KUKA KRL program: EPS_2_251727_MH2A_A_20260123013854.src

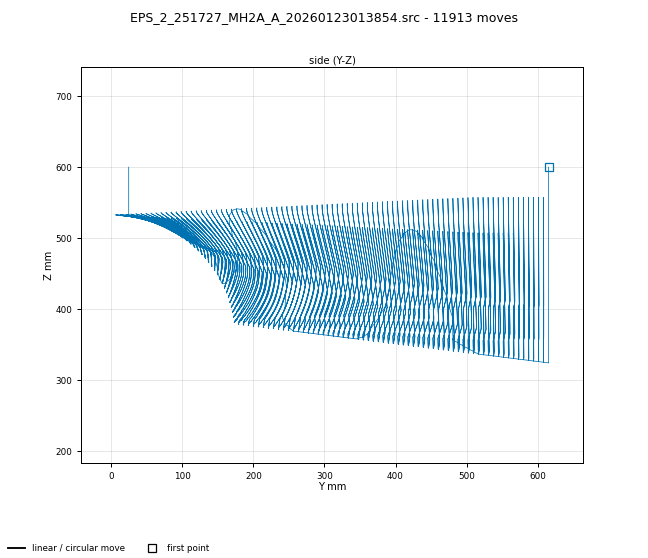
[picture p0: tool path of EPS_2_251727_MH2A_A_20260123013854.src, 11913 of 11915 moves have a stored position in this frame; points joined in program order, loops and branches not executed]
&ACCESS RVP
&REL 4
&COMMENT QRS 19112012
&PARAM EDITMASK = *
DEF PART()
EXT BAS (BAS_COMMAND :IN,REAL :IN )
INT I
BAS (#INITMOV,0 )

;KUKA QRS Post kuka4.cps  Date:22-06-2017 !

File_ID=2991

QRS_PRE_INIT()

;Init var - Until changes are made in qrs_pre_init
Outlet_Square_prg=0
Inlet_1_Square_prg=0
Inlet_2_Square_prg=0
Inlet_3_Square_prg=0
Inlet_4_Square_prg=0
Inlet_5_Square_prg=0

Outlet_1={X 0.000, Y 508.200, Z 408.000, B 0.000, E1 0.000 }
Inlet_1={X 0.000, Y 511.930, Z 358.000, B 0.000, E1 180.000 }
Outlet_1_type=299
Inlet_1_type=299
;QRS#1=Sidecore dimensions
;QRS#2=300-12" PVC SDR 35
;QRS#3=300-12" PVC SDR 35
;QRS#4=
;QRS#5=
;QRS#6=
;QRS#7=
;QRS#8=
;QRS#9=16M PSX
;QRS#10=16M PSX
;QRS#11=
;QRS#12=
;QRS#13=
;QRS#14=
;QRS#15=
;QRS#16=1220x127x838 2,75'
;QRS#17=EPS Height
;QRS#18=557,5
;QRS#19=*
;QRS#20= UPDATED VERSION 22-06-2017
;QRS#21=*
Outlet_Square=0150
Inlet_1_Square=0150
Inlet_2_Square=0
Inlet_3_Square=0
Inlet_4_Square=0
Inlet_5_Square=0
Mill_Square=1
Outlet_Square_Prg=206
Inlet_1_Square_prg=206

QRS_INIT()

$ADVANCE=5

; T1
PTP {E1 173.611,E2 173.611}
PTP {X 0,Y 615.501,A -85,B 0,C 180,E1 173.611,E2 173.611,E3 0,E4 0,E5 0,E6 0}
QRS_SPEED_INIT()
LIN {X 0,Y 615.501,Z 600,A -85,B 0,C 180,E1 173.611,E2 173.611,E3 0,E4 0,E5 0,E6 0} C_VEL
LIN {X 0,Y 615.501,Z 334.495,A -85,B 0,C 180,E1 173.611,E2 173.611} C_VEL
LIN {X 0,Y 615.501,Z 326.316,A -85,B 0,C 180,E1 173.611,E2 173.611} C_VEL
LIN {X 0,Y 615.486,Z 324.316,A -85,B 0,C 180,E1 173.425,E2 173.425} C_VEL
LIN {X 0,Y 615.496,Z 324.319,A -85,B 0,C 180,E1 170.801,E2 170.801} C_VEL
LIN {X 0,Y 615.493,Z 324.323,A -85,B 0,C 180,E1 168.139,E2 168.139} C_VEL
LIN {X 0,Y 615.481,Z 324.318,A -85,B 0,C 180,E1 165.451,E2 165.451} C_VEL
LIN {X 0,Y 615.494,Z 324.314,A -85,B 0,C 180,E1 162.73,E2 162.73} C_VEL
LIN {X 0,Y 615.494,Z 324.317,A -85,B 0,C 180,E1 159.967,E2 159.967} C_VEL
LIN {X 0,Y 615.493,Z 324.322,A -85,B 0,C 180,E1 157.156,E2 157.156} C_VEL
LIN {X 0,Y 615.5,Z 324.325,A -85,B 0,C 180,E1 154.285,E2 154.285} C_VEL
LIN {X 0,Y 615.479,Z 324.322,A -85,B 0,C 180,E1 151.552,E2 151.552} C_VEL
LIN {X 0,Y 615.487,Z 324.316,A -85,B 0,C 180,E1 148.915,E2 148.915} C_VEL
LIN {X 0,Y 615.49,Z 324.315,A -85,B 0,C 180,E1 145.978,E2 145.978} C_VEL
LIN {X 0,Y 615.487,Z 324.317,A -85,B 0,C 180,E1 143.064,E2 143.064} C_VEL
LIN {X 0,Y 615.495,Z 324.318,A -85,B 0,C 180,E1 140.25,E2 140.25} C_VEL
LIN {X 0,Y 615.487,Z 324.324,A -85,B 0,C 180,E1 137.647,E2 137.647} C_VEL
LIN {X 0,Y 615.487,Z 324.318,A -85,B 0,C 180,E1 134.931,E2 134.931} C_VEL
LIN {X 0,Y 615.481,Z 324.317,A -85,B 0,C 180,E1 132.079,E2 132.079} C_VEL
LIN {X 0,Y 615.496,Z 324.408,A -85,B 0,C 180,E1 131.473,E2 131.473} C_VEL
LIN {X 0,Y 615.484,Z 327.144,A -85,B 0,C 180,E1 128.905,E2 128.905} C_VEL
LIN {X 0,Y 615.494,Z 329.753,A -85,B 0,C 180,E1 126.425,E2 126.425} C_VEL
LIN {X 0,Y 615.496,Z 332.861,A -85,B 0,C 180,E1 123.535,E2 123.535} C_VEL
LIN {X 0,Y 615.48,Z 335.952,A -85,B 0,C 180,E1 120.92,E2 120.92} C_VEL
LIN {X 0,Y 615.491,Z 338.971,A -85,B 0,C 180,E1 118.451,E2 118.451} C_VEL
LIN {X 0,Y 615.499,Z 342.598,A -85,B 0,C 180,E1 115.571,E2 115.571} C_VEL
LIN {X 0,Y 615.482,Z 346.098,A -85,B 0,C 180,E1 112.845,E2 112.845} C_VEL
LIN {X 0,Y 615.484,Z 349.799,A -85,B 0,C 180,E1 110.033,E2 110.033} C_VEL
LIN {X 0,Y 615.478,Z 353.478,A -85,B 0,C 180,E1 107.271,E2 107.271} C_VEL
LIN {X 0,Y 615.481,Z 354.803,A -85,B 0,C 180,E1 106.298,E2 106.298} C_VEL
LIN {X 0,Y 615.497,Z 371.599,A -85,B 0,C 180,E1 106.003,E2 106.003} C_VEL
LIN {X 0,Y 615.49,Z 386.53,A -85,B 0,C 180,E1 105.608,E2 105.608} C_VEL
LIN {X 0,Y 615.48,Z 400.779,A -85,B 0,C 180,E1 105.099,E2 105.099} C_VEL
LIN {X 0,Y 615.482,Z 414.501,A -85,B 0,C 180,E1 104.473,E2 104.473} C_VEL
LIN {X 0,Y 615.496,Z 428.072,A -85,B 0,C 180,E1 103.706,E2 103.706} C_VEL
LIN {X 0,Y 615.496,Z 441.456,A -85,B 0,C 180,E1 102.782,E2 102.782} C_VEL
LIN {X 0,Y 615.495,Z 452.57,A -85,B 0,C 180,E1 101.861,E2 101.861} C_VEL
LIN {X 0,Y 615.493,Z 462.483,A -85,B 0,C 180,E1 100.89,E2 100.89} C_VEL
LIN {X 0,Y 615.495,Z 472.759,A -85,B 0,C 180,E1 99.696,E2 99.696} C_VEL
LIN {X 0,Y 615.49,Z 481.027,A -85,B 0,C 180,E1 98.537,E2 98.537} C_VEL
LIN {X 0,Y 615.491,Z 488.782,A -85,B 0,C 180,E1 97.216,E2 97.216} C_VEL
LIN {X 0,Y 615.499,Z 494.947,A -85,B 0,C 180,E1 95.899,E2 95.899} C_VEL
LIN {X 0,Y 615.489,Z 499.716,A -85,B 0,C 180,E1 94.585,E2 94.585} C_VEL
LIN {X 0,Y 615.491,Z 503.22,A -85,B 0,C 180,E1 93.273,E2 93.273} C_VEL
LIN {X 0,Y 615.5,Z 505.539,A -85,B 0,C 180,E1 91.963,E2 91.963} C_VEL
LIN {X 0,Y 615.491,Z 506.728,A -85,B 0,C 180,E1 90.655,E2 90.655} C_VEL
LIN {X 0,Y 615.492,Z 506.751,A -85,B 0,C 180,E1 89.346,E2 89.346} C_VEL
LIN {X 0,Y 615.5,Z 505.646,A -85,B 0,C 180,E1 88.037,E2 88.037} C_VEL
LIN {X 0,Y 615.494,Z 503.416,A -85,B 0,C 180,E1 86.727,E2 86.727} C_VEL
LIN {X 0,Y 615.49,Z 500.006,A -85,B 0,C 180,E1 85.416,E2 85.416} C_VEL
LIN {X 0,Y 615.499,Z 495.337,A -85,B 0,C 180,E1 84.102,E2 84.102} C_VEL
LIN {X 0,Y 615.49,Z 489.273,A -85,B 0,C 180,E1 82.785,E2 82.785} C_VEL
LIN {X 0,Y 615.493,Z 481.634,A -85,B 0,C 180,E1 81.464,E2 81.464} C_VEL
LIN {X 0,Y 615.496,Z 473.452,A -85,B 0,C 180,E1 80.304,E2 80.304} C_VEL
LIN {X 0,Y 615.495,Z 463.338,A -85,B 0,C 180,E1 79.109,E2 79.109} C_VEL
LIN {X 0,Y 615.497,Z 451.686,A -85,B 0,C 180,E1 77.973,E2 77.973} C_VEL
LIN {X 0,Y 615.498,Z 440.416,A -85,B 0,C 180,E1 77.051,E2 77.051} C_VEL
LIN {X 0,Y 615.498,Z 428.177,A -85,B 0,C 180,E1 76.211,E2 76.211} C_VEL
LIN {X 0,Y 615.49,Z 414.78,A -85,B 0,C 180,E1 75.451,E2 75.451} C_VEL
LIN {X 0,Y 615.478,Z 400.916,A -85,B 0,C 180,E1 74.816,E2 74.816} C_VEL
LIN {X 0,Y 615.496,Z 386.702,A -85,B 0,C 180,E1 74.308,E2 74.308} C_VEL
LIN {X 0,Y 615.494,Z 372.662,A -85,B 0,C 180,E1 73.932,E2 73.932} C_VEL
LIN {X 0,Y 615.483,Z 357.246,A -85,B 0,C 180,E1 73.652,E2 73.652} C_VEL
LIN {X 0,Y 615.483,Z 354.79,A -85,B 0,C 180,E1 73.603,E2 73.603} C_VEL
LIN {X 0,Y 615.487,Z 351.76,A -85,B 0,C 180,E1 71.354,E2 71.354} C_VEL
LIN {X 0,Y 615.485,Z 348.062,A -85,B 0,C 180,E1 68.568,E2 68.568} C_VEL
LIN {X 0,Y 615.48,Z 344.375,A -85,B 0,C 180,E1 65.728,E2 65.728} C_VEL
LIN {X 0,Y 615.48,Z 340.845,A -85,B 0,C 180,E1 62.957,E2 62.957} C_VEL
LIN {X 0,Y 615.477,Z 337.437,A -85,B 0,C 180,E1 60.207,E2 60.207} C_VEL
LIN {X 0,Y 615.493,Z 334.207,A -85,B 0,C 180,E1 57.543,E2 57.543} C_VEL
LIN {X 0,Y 615.497,Z 331.577,A -85,B 0,C 180,E1 55.186,E2 55.186} C_VEL
LIN {X 0,Y 615.493,Z 328.991,A -85,B 0,C 180,E1 52.759,E2 52.759} C_VEL
LIN {X 0,Y 615.49,Z 325.998,A -85,B 0,C 180,E1 49.911,E2 49.911} C_VEL
LIN {X 0,Y 615.497,Z 324.507,A -85,B 0,C 180,E1 48.527,E2 48.527} C_VEL
LIN {X 0,Y 615.491,Z 324.317,A -85,B 0,C 180,E1 45.851,E2 45.851} C_VEL
LIN {X 0,Y 615.483,Z 324.317,A -85,B 0,C 180,E1 43.047,E2 43.047} C_VEL
LIN {X 0,Y 615.481,Z 324.322,A -85,B 0,C 180,E1 40.607,E2 40.607} C_VEL
LIN {X 0,Y 615.485,Z 324.323,A -85,B 0,C 180,E1 38.012,E2 38.012} C_VEL
LIN {X 0,Y 615.481,Z 324.317,A -85,B 0,C 180,E1 35.616,E2 35.616} C_VEL
LIN {X 0,Y 615.489,Z 324.327,A -85,B 0,C 180,E1 33.236,E2 33.236} C_VEL
LIN {X 0,Y 615.49,Z 324.315,A -85,B 0,C 180,E1 30.92,E2 30.92} C_VEL
LIN {X 0,Y 615.479,Z 324.323,A -85,B 0,C 180,E1 28.45,E2 28.45} C_VEL
LIN {X 0,Y 615.498,Z 324.324,A -85,B 0,C 180,E1 25.715,E2 25.715} C_VEL
LIN {X 0,Y 615.494,Z 324.32,A -85,B 0,C 180,E1 22.844,E2 22.844} C_VEL
LIN {X 0,Y 615.493,Z 324.316,A -85,B 0,C 180,E1 20.033,E2 20.033} C_VEL
LIN {X 0,Y 615.493,Z 324.314,A -85,B 0,C 180,E1 17.27,E2 17.27} C_VEL
LIN {X 0,Y 615.481,Z 324.319,A -85,B 0,C 180,E1 14.549,E2 14.549} C_VEL
LIN {X 0,Y 615.492,Z 324.324,A -85,B 0,C 180,E1 11.861,E2 11.861} C_VEL
LIN {X 0,Y 615.496,Z 324.318,A -85,B 0,C 180,E1 9.199,E2 9.199} C_VEL
LIN {X 0,Y 615.487,Z 324.316,A -85,B 0,C 180,E1 6.557,E2 6.557} C_VEL
LIN {X 0,Y 615.48,Z 324.32,A -85,B 0,C 180,E1 3.929,E2 3.929} C_VEL
LIN {X 0,Y 615.495,Z 324.326,A -85,B 0,C 180,E1 1.309,E2 1.309} C_VEL
LIN {X 0,Y 615.487,Z 324.318,A -85,B 0,C 180,E1 -1.309,E2 -1.309} C_VEL
LIN {X 0,Y 615.478,Z 324.318,A -85,B 0,C 180,E1 -3.928,E2 -3.928} C_VEL
LIN {X 0,Y 615.486,Z 324.321,A -85,B 0,C 180,E1 -6.58,E2 -6.58} C_VEL
LIN {X 0,Y 615.489,Z 324.323,A -85,B 0,C 180,E1 -9.199,E2 -9.199} C_VEL
LIN {X 0,Y 615.477,Z 324.319,A -85,B 0,C 180,E1 -11.861,E2 -11.861} C_VEL
LIN {X 0,Y 615.481,Z 324.317,A -85,B 0,C 180,E1 -14.549,E2 -14.549} C_VEL
LIN {X 0,Y 615.493,Z 324.319,A -85,B 0,C 180,E1 -17.27,E2 -17.27} C_VEL
LIN {X 0,Y 615.493,Z 324.326,A -85,B 0,C 180,E1 -20.033,E2 -20.033} C_VEL
LIN {X 0,Y 615.483,Z 324.323,A -85,B 0,C 180,E1 -22.845,E2 -22.845} C_VEL
LIN {X 0,Y 615.476,Z 324.319,A -85,B 0,C 180,E1 -25.567,E2 -25.567} C_VEL
LIN {X 0,Y 615.491,Z 324.32,A -85,B 0,C 180,E1 -27.915,E2 -27.915} C_VEL
LIN {X 0,Y 615.492,Z 324.316,A -85,B 0,C 180,E1 -30.16,E2 -30.16} C_VEL
LIN {X 0,Y 615.477,Z 324.323,A -85,B 0,C 180,E1 -32.458,E2 -32.458} C_VEL
LIN {X 0,Y 615.491,Z 324.317,A -85,B 0,C 180,E1 -34.815,E2 -34.815} C_VEL
LIN {X 0,Y 615.479,Z 324.319,A -85,B 0,C 180,E1 -37.243,E2 -37.243} C_VEL
LIN {X 0,Y 615.483,Z 324.321,A -85,B 0,C 180,E1 -40.089,E2 -40.089} C_VEL
LIN {X 0,Y 615.477,Z 324.319,A -85,B 0,C 180,E1 -42.354,E2 -42.354} C_VEL
LIN {X 0,Y 615.479,Z 324.318,A -85,B 0,C 180,E1 -45.069,E2 -45.069} C_VEL
LIN {X 0,Y 615.485,Z 324.318,A -85,B 0,C 180,E1 -47.92,E2 -47.92} C_VEL
LIN {X 0,Y 615.499,Z 324.463,A -85,B 0,C 180,E1 -48.717,E2 -48.717} C_VEL
LIN {X 0,Y 615.482,Z 331.995,A -85,B 0,C 180,E1 -51.515,E2 -51.515} C_VEL
LIN {X 0,Y 615.48,Z 339.577,A -85,B 0,C 180,E1 -54.167,E2 -54.167} C_VEL
LIN {X 0,Y 615.485,Z 347.271,A -85,B 0,C 180,E1 -56.764,E2 -56.764} C_VEL
LIN {X 0,Y 615.496,Z 355.427,A -85,B 0,C 180,E1 -59.462,E2 -59.462} C_VEL
LIN {X 0,Y 615.495,Z 364.738,A -85,B 0,C 180,E1 -62.455,E2 -62.455} C_VEL
LIN {X 0,Y 615.493,Z 374.043,A -85,B 0,C 180,E1 -65.369,E2 -65.369} C_VEL
LIN {X 0,Y 615.489,Z 383.349,A -85,B 0,C 180,E1 -68.217,E2 -68.217} C_VEL
LIN {X 0,Y 615.484,Z 392.643,A -85,B 0,C 180,E1 -71.009,E2 -71.009} C_VEL
LIN {X 0,Y 615.488,Z 401.469,A -85,B 0,C 180,E1 -73.618,E2 -73.618} C_VEL
LIN {X 0,Y 615.493,Z 417.381,A -85,B 0,C 180,E1 -73.865,E2 -73.865} C_VEL
LIN {X 0,Y 615.497,Z 432.296,A -85,B 0,C 180,E1 -74.223,E2 -74.223} C_VEL
LIN {X 0,Y 615.478,Z 446.433,A -85,B 0,C 180,E1 -74.689,E2 -74.689} C_VEL
LIN {X 0,Y 615.496,Z 460.364,A -85,B 0,C 180,E1 -75.282,E2 -75.282} C_VEL
LIN {X 0,Y 615.499,Z 473.674,A -85,B 0,C 180,E1 -75.986,E2 -75.986} C_VEL
LIN {X 0,Y 615.498,Z 486.319,A -85,B 0,C 180,E1 -76.799,E2 -76.799} C_VEL
LIN {X 0,Y 615.496,Z 497.297,A -85,B 0,C 180,E1 -77.638,E2 -77.638} C_VEL
LIN {X 0,Y 615.497,Z 508.357,A -85,B 0,C 180,E1 -78.641,E2 -78.641} C_VEL
LIN {X 0,Y 615.496,Z 519.071,A -85,B 0,C 180,E1 -79.806,E2 -79.806} C_VEL
LIN {X 0,Y 615.495,Z 527.99,A -85,B 0,C 180,E1 -80.967,E2 -80.967} C_VEL
LIN {X 0,Y 615.492,Z 535.395,A -85,B 0,C 180,E1 -82.125,E2 -82.125} C_VEL
LIN {X 0,Y 615.491,Z 542.274,A -85,B 0,C 180,E1 -83.444,E2 -83.444} C_VEL
LIN {X 0,Y 615.491,Z 547.667,A -85,B 0,C 180,E1 -84.759,E2 -84.759} C_VEL
LIN {X 0,Y 615.491,Z 551.742,A -85,B 0,C 180,E1 -86.072,E2 -86.072} C_VEL
LIN {X 0,Y 615.496,Z 554.6,A -85,B 0,C 180,E1 -87.382,E2 -87.382} C_VEL
LIN {X 0,Y 615.493,Z 556.307,A -85,B 0,C 180,E1 -88.692,E2 -88.692} C_VEL
LIN {X 0,Y 615.491,Z 556.889,A -85,B 0,C 180,E1 -90,E2 -90} C_VEL
LIN {X 0,Y 615.493,Z 556.306,A -85,B 0,C 180,E1 -91.309,E2 -91.309} C_VEL
LIN {X 0,Y 615.496,Z 554.599,A -85,B 0,C 180,E1 -92.618,E2 -92.618} C_VEL
LIN {X 0,Y 615.491,Z 551.74,A -85,B 0,C 180,E1 -93.929,E2 -93.929} C_VEL
LIN {X 0,Y 615.491,Z 547.665,A -85,B 0,C 180,E1 -95.241,E2 -95.241} C_VEL
LIN {X 0,Y 615.491,Z 542.153,A -85,B 0,C 180,E1 -96.581,E2 -96.581} C_VEL
LIN {X 0,Y 615.492,Z 535.391,A -85,B 0,C 180,E1 -97.876,E2 -97.876} C_VEL
LIN {X 0,Y 615.495,Z 526.807,A -85,B 0,C 180,E1 -99.199,E2 -99.199} C_VEL
LIN {X 0,Y 615.494,Z 517.665,A -85,B 0,C 180,E1 -100.361,E2 -100.361} C_VEL
LIN {X 0,Y 615.497,Z 508.351,A -85,B 0,C 180,E1 -101.36,E2 -101.36} C_VEL
LIN {X 0,Y 615.496,Z 497.29,A -85,B 0,C 180,E1 -102.363,E2 -102.363} C_VEL
LIN {X 0,Y 615.498,Z 485.149,A -85,B 0,C 180,E1 -103.285,E2 -103.285} C_VEL
LIN {X 0,Y 615.498,Z 472.404,A -85,B 0,C 180,E1 -104.09,E2 -104.09} C_VEL
LIN {X 0,Y 615.496,Z 458.605,A -85,B 0,C 180,E1 -104.803,E2 -104.803} C_VEL
LIN {X 0,Y 615.48,Z 444.176,A -85,B 0,C 180,E1 -105.396,E2 -105.396} C_VEL
LIN {X 0,Y 615.496,Z 429.239,A -85,B 0,C 180,E1 -105.863,E2 -105.863} C_VEL
LIN {X 0,Y 615.491,Z 413.838,A -85,B 0,C 180,E1 -106.201,E2 -106.201} C_VEL
LIN {X 0,Y 615.488,Z 401.413,A -85,B 0,C 180,E1 -106.399,E2 -106.399} C_VEL
LIN {X 0,Y 615.484,Z 392.641,A -85,B 0,C 180,E1 -108.992,E2 -108.992} C_VEL
LIN {X 0,Y 615.489,Z 383.348,A -85,B 0,C 180,E1 -111.784,E2 -111.784} C_VEL
LIN {X 0,Y 615.493,Z 374.041,A -85,B 0,C 180,E1 -114.631,E2 -114.631} C_VEL
LIN {X 0,Y 615.494,Z 364.736,A -85,B 0,C 180,E1 -117.545,E2 -117.545} C_VEL
LIN {X 0,Y 615.496,Z 355.425,A -85,B 0,C 180,E1 -120.539,E2 -120.539} C_VEL
LIN {X 0,Y 615.485,Z 347.269,A -85,B 0,C 180,E1 -123.237,E2 -123.237} C_VEL
LIN {X 0,Y 615.48,Z 339.58,A -85,B 0,C 180,E1 -125.833,E2 -125.833} C_VEL
LIN {X 0,Y 615.485,Z 331.993,A -85,B 0,C 180,E1 -128.486,E2 -128.486} C_VEL
LIN {X 0,Y 615.498,Z 324.463,A -85,B 0,C 180,E1 -131.284,E2 -131.284} C_VEL
LIN {X 0,Y 615.491,Z 324.324,A -85,B 0,C 180,E1 -133.998,E2 -133.998} C_VEL
LIN {X 0,Y 615.483,Z 324.323,A -85,B 0,C 180,E1 -136.953,E2 -136.953} C_VEL
LIN {X 0,Y 615.482,Z 324.317,A -85,B 0,C 180,E1 -139.393,E2 -139.393} C_VEL
LIN {X 0,Y 615.493,Z 324.32,A -85,B 0,C 180,E1 -141.988,E2 -141.988} C_VEL
LIN {X 0,Y 615.487,Z 324.319,A -85,B 0,C 180,E1 -144.384,E2 -144.384} C_VEL
LIN {X 0,Y 615.481,Z 324.319,A -85,B 0,C 180,E1 -146.763,E2 -146.763} C_VEL
LIN {X 0,Y 615.493,Z 324.32,A -85,B 0,C 180,E1 -149.081,E2 -149.081} C_VEL
LIN {X 0,Y 615.478,Z 324.318,A -85,B 0,C 180,E1 -151.552,E2 -151.552} C_VEL
LIN {X 0,Y 615.477,Z 324.321,A -85,B 0,C 180,E1 -154.284,E2 -154.284} C_VEL
LIN {X 0,Y 615.474,Z 324.32,A -85,B 0,C 180,E1 -156.443,E2 -156.443} C_VEL
LIN {X 0,Y 615.498,Z 324.323,A -85,B 0,C 180,E1 -158.569,E2 -158.569} C_VEL
LIN {X 0,Y 615.486,Z 324.324,A -85,B 0,C 180,E1 -161.396,E2 -161.396} C_VEL
LIN {X 0,Y 615.482,Z 324.318,A -85,B 0,C 180,E1 -164.095,E2 -164.095} C_VEL
LIN {X 0,Y 615.494,Z 324.314,A -85,B 0,C 180,E1 -166.799,E2 -166.799} C_VEL
LIN {X 0,Y 615.494,Z 324.318,A -85,B 0,C 180,E1 -169.473,E2 -169.473} C_VEL
LIN {X 0,Y 615.49,Z 324.325,A -85,B 0,C 180,E1 -172.124,E2 -172.124} C_VEL
LIN {X 0,Y 615.487,Z 324.317,A -85,B 0,C 180,E1 -174.759,E2 -174.759} C_VEL
LIN {X 0,Y 615.491,Z 324.315,A -85,B 0,C 180,E1 -177.382,E2 -177.382} C_VEL
LIN {X 0,Y 615.486,Z 324.323,A -85,B 0,C 180,E1 -180,E2 -180} C_VEL
LIN {X 0,Y 615.496,Z 324.319,A -85,B 0,C 180,E1 -182.618,E2 -182.618} C_VEL
LIN {X 0,Y 615.487,Z 324.316,A -85,B 0,C 180,E1 -185.241,E2 -185.241} C_VEL
LIN {X 0,Y 615.486,Z 324.316,A -85,B 0,C 180,E1 -186.575,E2 -186.575} C_VEL
LIN {X 0,Y 614.812,Z 324.469,A -85,B 0,C 180,E1 -187.121,E2 -187.121} C_VEL
LIN {X 0,Y 611.984,Z 324.877,A -85,B 0,C 180,E1 -188.007,E2 -188.007} C_VEL
LIN {X 0,Y 609.595,Z 325.188,A -85,B 0,C 180,E1 -188.72,E2 -188.72} C_VEL
LIN {X 0,Y 608.556,Z 325.307,A -85,B 0,C 180,E1 -189.269,E2 -189.269} C_VEL
LIN {X 0,Y 608.464,Z 325.316,A -85,B 0,C 180,E1 -189.455,E2 -189.455} C_VEL
LIN {X 0,Y 608.466,Z 325.321,A -85,B 0,C 180,E1 -192,E2 -192} C_VEL
LIN {X 0,Y 608.474,Z 325.316,A -85,B 0,C 180,E1 -194.721,E2 -194.721} C_VEL
LIN {X 0,Y 608.458,Z 325.316,A -85,B 0,C 180,E1 -197.476,E2 -197.476} C_VEL
LIN {X 0,Y 608.461,Z 325.315,A -85,B 0,C 180,E1 -200.274,E2 -200.274} C_VEL
LIN {X 0,Y 608.462,Z 325.319,A -85,B 0,C 180,E1 -202.476,E2 -202.476} C_VEL
LIN {X 0,Y 608.458,Z 325.318,A -85,B 0,C 180,E1 -204.571,E2 -204.571} C_VEL
LIN {X 0,Y 608.485,Z 325.319,A -85,B 0,C 180,E1 -207.208,E2 -207.208} C_VEL
LIN {X 0,Y 608.47,Z 325.317,A -85,B 0,C 180,E1 -209.971,E2 -209.971} C_VEL
LIN {X 0,Y 608.459,Z 325.317,A -85,B 0,C 180,E1 -212.88,E2 -212.88} C_VEL
LIN {X 0,Y 608.443,Z 325.319,A -85,B 0,C 180,E1 -215.278,E2 -215.278} C_VEL
LIN {X 0,Y 608.467,Z 325.319,A -85,B 0,C 180,E1 -217.746,E2 -217.746} C_VEL
LIN {X 0,Y 608.448,Z 325.318,A -85,B 0,C 180,E1 -220.328,E2 -220.328} C_VEL
LIN {X 0,Y 608.45,Z 325.318,A -85,B 0,C 180,E1 -222.96,E2 -222.96} C_VEL
LIN {X 0,Y 608.46,Z 325.319,A -85,B 0,C 180,E1 -225.736,E2 -225.736} C_VEL
LIN {X 0,Y 608.461,Z 325.316,A -85,B 0,C 180,E1 -227.938,E2 -227.938} C_VEL
LIN {X 0,Y 608.445,Z 325.62,A -85,B 0,C 180,E1 -228.822,E2 -228.822} C_VEL
LIN {X 0,Y 608.438,Z 328.355,A -85,B 0,C 180,E1 -231.409,E2 -231.409} C_VEL
LIN {X 0,Y 608.451,Z 331.034,A -85,B 0,C 180,E1 -233.954,E2 -233.954} C_VEL
LIN {X 0,Y 608.456,Z 333.56,A -85,B 0,C 180,E1 -236.329,E2 -236.329} C_VEL
LIN {X 0,Y 608.449,Z 336.318,A -85,B 0,C 180,E1 -238.732,E2 -238.732} C_VEL
LIN {X 0,Y 608.427,Z 339.55,A -85,B 0,C 180,E1 -241.388,E2 -241.388} C_VEL
LIN {X 0,Y 608.428,Z 343.171,A -85,B 0,C 180,E1 -244.288,E2 -244.288} C_VEL
LIN {X 0,Y 608.413,Z 346.478,A -85,B 0,C 180,E1 -246.874,E2 -246.874} C_VEL
LIN {X 0,Y 608.427,Z 350.194,A -85,B 0,C 180,E1 -249.724,E2 -249.724} C_VEL
LIN {X 0,Y 608.41,Z 353.911,A -85,B 0,C 180,E1 -252.522,E2 -252.522} C_VEL
LIN {X 0,Y 608.441,Z 355.245,A -85,B 0,C 180,E1 -253.516,E2 -253.516} C_VEL
LIN {X 0,Y 608.671,Z 370.922,A -85,B 0,C 180,E1 -253.796,E2 -253.796} C_VEL
LIN {X 0,Y 608.641,Z 385.226,A -85,B 0,C 180,E1 -254.169,E2 -254.169} C_VEL
LIN {X 0,Y 608.614,Z 399.728,A -85,B 0,C 180,E1 -254.683,E2 -254.683} C_VEL
LIN {X 0,Y 608.572,Z 412.933,A -85,B 0,C 180,E1 -255.282,E2 -255.282} C_VEL
LIN {X 0,Y 608.565,Z 426.697,A -85,B 0,C 180,E1 -256.05,E2 -256.05} C_VEL
LIN {X 0,Y 608.548,Z 439.235,A -85,B 0,C 180,E1 -256.9,E2 -256.9} C_VEL
LIN {X 0,Y 608.522,Z 450.755,A -85,B 0,C 180,E1 -257.832,E2 -257.832} C_VEL
LIN {X 0,Y 608.483,Z 460.964,A -85,B 0,C 180,E1 -258.807,E2 -258.807} C_VEL
LIN {X 0,Y 608.48,Z 470.293,A -85,B 0,C 180,E1 -259.855,E2 -259.855} C_VEL
LIN {X 0,Y 608.447,Z 479.108,A -85,B 0,C 180,E1 -261.029,E2 -261.029} C_VEL
LIN {X 0,Y 608.457,Z 485.478,A -85,B 0,C 180,E1 -262.033,E2 -262.033} C_VEL
LIN {X 0,Y 608.445,Z 492.628,A -85,B 0,C 180,E1 -263.397,E2 -263.397} C_VEL
LIN {X 0,Y 608.435,Z 497.992,A -85,B 0,C 180,E1 -264.698,E2 -264.698} C_VEL
LIN {X 0,Y 608.432,Z 502.166,A -85,B 0,C 180,E1 -266.026,E2 -266.026} C_VEL
LIN {X 0,Y 608.421,Z 505.109,A -85,B 0,C 180,E1 -267.351,E2 -267.351} C_VEL
LIN {X 0,Y 608.444,Z 506.88,A -85,B 0,C 180,E1 -268.676,E2 -268.676} C_VEL
LIN {X 0,Y 608.432,Z 507.495,A -85,B 0,C 180,E1 -270,E2 -270} C_VEL
LIN {X 0,Y 608.446,Z 506.944,A -85,B 0,C 180,E1 -271.323,E2 -271.323} C_VEL
LIN {X 0,Y 608.424,Z 505.26,A -85,B 0,C 180,E1 -272.648,E2 -272.648} C_VEL
LIN {X 0,Y 608.431,Z 502.409,A -85,B 0,C 180,E1 -273.974,E2 -273.974} C_VEL
LIN {X 0,Y 608.435,Z 498.329,A -85,B 0,C 180,E1 -275.302,E2 -275.302} C_VEL
LIN {X 0,Y 608.445,Z 492.923,A -85,B 0,C 180,E1 -276.633,E2 -276.633} C_VEL
LIN {X 0,Y 608.456,Z 486.025,A -85,B 0,C 180,E1 -277.967,E2 -277.967} C_VEL
LIN {X 0,Y 608.466,Z 478.593,A -85,B 0,C 180,E1 -279.138,E2 -279.138} C_VEL
LIN {X 0,Y 608.476,Z 469.665,A -85,B 0,C 180,E1 -280.313,E2 -280.313} C_VEL
LIN {X 0,Y 608.495,Z 458.95,A -85,B 0,C 180,E1 -281.492,E2 -281.492} C_VEL
LIN {X 0,Y 608.513,Z 446.909,A -85,B 0,C 180,E1 -282.591,E2 -282.591} C_VEL
LIN {X 0,Y 608.543,Z 434.622,A -85,B 0,C 180,E1 -283.524,E2 -283.524} C_VEL
LIN {X 0,Y 608.579,Z 421.067,A -85,B 0,C 180,E1 -284.375,E2 -284.375} C_VEL
LIN {X 0,Y 608.592,Z 407.776,A -85,B 0,C 180,E1 -285.06,E2 -285.06} C_VEL
LIN {X 0,Y 608.615,Z 393.114,A -85,B 0,C 180,E1 -285.659,E2 -285.659} C_VEL
LIN {X 0,Y 608.664,Z 377.543,A -85,B 0,C 180,E1 -286.138,E2 -286.138} C_VEL
LIN {X 0,Y 608.67,Z 362.055,A -85,B 0,C 180,E1 -286.466,E2 -286.466} C_VEL
LIN {X 0,Y 608.428,Z 355.25,A -85,B 0,C 180,E1 -286.571,E2 -286.571} C_VEL
LIN {X 0,Y 608.42,Z 352.173,A -85,B 0,C 180,E1 -288.87,E2 -288.87} C_VEL
LIN {X 0,Y 608.41,Z 348.454,A -85,B 0,C 180,E1 -291.693,E2 -291.693} C_VEL
LIN {X 0,Y 608.417,Z 344.735,A -85,B 0,C 180,E1 -294.572,E2 -294.572} C_VEL
LIN {X 0,Y 608.427,Z 341.417,A -85,B 0,C 180,E1 -297.197,E2 -297.197} C_VEL
LIN {X 0,Y 608.442,Z 337.999,A -85,B 0,C 180,E1 -299.967,E2 -299.967} C_VEL
LIN {X 0,Y 608.435,Z 334.935,A -85,B 0,C 180,E1 -302.518,E2 -302.518} C_VEL
LIN {X 0,Y 608.448,Z 331.955,A -85,B 0,C 180,E1 -305.277,E2 -305.277} C_VEL
LIN {X 0,Y 608.454,Z 329.334,A -85,B 0,C 180,E1 -307.747,E2 -307.747} C_VEL
LIN {X 0,Y 608.442,Z 326.637,A -85,B 0,C 180,E1 -310.328,E2 -310.328} C_VEL
LIN {X 0,Y 608.47,Z 325.54,A -85,B 0,C 180,E1 -311.343,E2 -311.343} C_VEL
LIN {X 0,Y 608.468,Z 325.315,A -85,B 0,C 180,E1 -313.869,E2 -313.869} C_VEL
LIN {X 0,Y 608.467,Z 325.315,A -85,B 0,C 180,E1 -316.691,E2 -316.691} C_VEL
LIN {X 0,Y 608.452,Z 325.319,A -85,B 0,C 180,E1 -318.823,E2 -318.823} C_VEL
LIN {X 0,Y 608.472,Z 325.314,A -85,B 0,C 180,E1 -321.412,E2 -321.412} C_VEL
LIN {X 0,Y 608.479,Z 325.316,A -85,B 0,C 180,E1 -323.95,E2 -323.95} C_VEL
LIN {X 0,Y 608.448,Z 325.319,A -85,B 0,C 180,E1 -326.328,E2 -326.328} C_VEL
LIN {X 0,Y 608.477,Z 325.315,A -85,B 0,C 180,E1 -328.727,E2 -328.727} C_VEL
LIN {X 0,Y 608.472,Z 325.32,A -85,B 0,C 180,E1 -331.38,E2 -331.38} C_VEL
LIN {X 0,Y 608.448,Z 325.319,A -85,B 0,C 180,E1 -333.964,E2 -333.964} C_VEL
LIN {X 0,Y 608.467,Z 325.318,A -85,B 0,C 180,E1 -336.155,E2 -336.155} C_VEL
LIN {X 0,Y 608.468,Z 325.315,A -85,B 0,C 180,E1 -338.308,E2 -338.308} C_VEL
LIN {X 0,Y 608.453,Z 325.317,A -85,B 0,C 180,E1 -341.13,E2 -341.13} C_VEL
LIN {X 0,Y 608.458,Z 325.317,A -85,B 0,C 180,E1 -343.906,E2 -343.906} C_VEL
LIN {X 0,Y 608.468,Z 325.319,A -85,B 0,C 180,E1 -346.644,E2 -346.644} C_VEL
LIN {X 0,Y 608.467,Z 325.318,A -85,B 0,C 180,E1 -349.35,E2 -349.35} C_VEL
LIN {X 0,Y 608.472,Z 325.315,A -85,B 0,C 180,E1 -352.033,E2 -352.033} C_VEL
LIN {X 0,Y 608.467,Z 325.315,A -85,B 0,C 180,E1 -354.698,E2 -354.698} C_VEL
LIN {X 0,Y 608.486,Z 325.317,A -85,B 0,C 180,E1 -357.352,E2 -357.352} C_VEL
LIN {X 0,Y 608.474,Z 325.317,A -85,B 0,C 180,E1 -360,E2 -360} C_VEL
LIN {X 0,Y 608.481,Z 325.313,A -85,B 0,C 180,E1 -362.648,E2 -362.648} C_VEL
LIN {X 0,Y 608.47,Z 325.315,A -85,B 0,C 180,E1 -365.302,E2 -365.302} C_VEL
LIN {X 0,Y 608.482,Z 325.318,A -85,B 0,C 180,E1 -367.967,E2 -367.967} C_VEL
LIN {X 0,Y 608.473,Z 325.32,A -85,B 0,C 180,E1 -370.959,E2 -370.959} C_VEL
LIN {X 0,Y 608.471,Z 325.315,A -85,B 0,C 180,E1 -373.356,E2 -373.356} C_VEL
LIN {X 0,Y 608.46,Z 325.316,A -85,B 0,C 180,E1 -376.094,E2 -376.094} C_VEL
LIN {X 0,Y 608.457,Z 325.318,A -85,B 0,C 180,E1 -378.87,E2 -378.87} C_VEL
LIN {X 0,Y 608.478,Z 325.318,A -85,B 0,C 180,E1 -381.691,E2 -381.691} C_VEL
LIN {X 0,Y 608.46,Z 325.322,A -85,B 0,C 180,E1 -384.571,E2 -384.571} C_VEL
LIN {X 0,Y 608.455,Z 325.321,A -85,B 0,C 180,E1 -387.518,E2 -387.518} C_VEL
LIN {X 0,Y 608.47,Z 325.315,A -85,B 0,C 180,E1 -389.973,E2 -389.973} C_VEL
LIN {X 0,Y 608.454,Z 325.319,A -85,B 0,C 180,E1 -392.522,E2 -392.522} C_VEL
LIN {X 0,Y 608.446,Z 325.324,A -85,B 0,C 180,E1 -395.277,E2 -395.277} C_VEL
LIN {X 0,Y 608.473,Z 325.32,A -85,B 0,C 180,E1 -398.242,E2 -398.242} C_VEL
LIN {X 0,Y 608.464,Z 325.32,A -85,B 0,C 180,E1 -401.176,E2 -401.176} C_VEL
LIN {X 0,Y 608.474,Z 325.315,A -85,B 0,C 180,E1 -403.869,E2 -403.869} C_VEL
LIN {X 0,Y 608.482,Z 325.314,A -85,B 0,C 180,E1 -406.69,E2 -406.69} C_VEL
LIN {X 0,Y 608.48,Z 325.421,A -85,B 0,C 180,E1 -408.522,E2 -408.522} C_VEL
LIN {X 0,Y 608.506,Z 331.117,A -85,B 0,C 180,E1 -410.698,E2 -410.698} C_VEL
LIN {X 0,Y 608.516,Z 338.969,A -85,B 0,C 180,E1 -413.502,E2 -413.502} C_VEL
LIN {X 0,Y 608.504,Z 347.294,A -85,B 0,C 180,E1 -416.332,E2 -416.332} C_VEL
LIN {X 0,Y 608.507,Z 355.544,A -85,B 0,C 180,E1 -419.094,E2 -419.094} C_VEL
LIN {X 0,Y 608.476,Z 363.652,A -85,B 0,C 180,E1 -421.735,E2 -421.735} C_VEL
LIN {X 0,Y 608.475,Z 371.648,A -85,B 0,C 180,E1 -424.278,E2 -424.278} C_VEL
LIN {X 0,Y 608.464,Z 379.997,A -85,B 0,C 180,E1 -426.877,E2 -426.877} C_VEL
LIN {X 0,Y 608.468,Z 387.998,A -85,B 0,C 180,E1 -429.321,E2 -429.321} C_VEL
LIN {X 0,Y 608.449,Z 397.51,A -85,B 0,C 180,E1 -432.176,E2 -432.176} C_VEL
LIN {X 0,Y 608.462,Z 401.723,A -85,B 0,C 180,E1 -433.427,E2 -433.427} C_VEL
LIN {X 0,Y 608.678,Z 412.21,A -85,B 0,C 180,E1 -433.582,E2 -433.582} C_VEL
LIN {X 0,Y 608.656,Z 427.724,A -85,B 0,C 180,E1 -433.912,E2 -433.912} C_VEL
LIN {X 0,Y 608.629,Z 443.058,A -85,B 0,C 180,E1 -434.384,E2 -434.384} C_VEL
LIN {X 0,Y 608.615,Z 456.763,A -85,B 0,C 180,E1 -434.941,E2 -434.941} C_VEL
LIN {X 0,Y 608.591,Z 470.862,A -85,B 0,C 180,E1 -435.659,E2 -435.659} C_VEL
LIN {X 0,Y 608.543,Z 483.946,A -85,B 0,C 180,E1 -436.476,E2 -436.476} C_VEL
LIN {X 0,Y 608.512,Z 496.346,A -85,B 0,C 180,E1 -437.409,E2 -437.409} C_VEL
LIN {X 0,Y 608.496,Z 506.751,A -85,B 0,C 180,E1 -438.339,E2 -438.339} C_VEL
LIN {X 0,Y 608.477,Z 516.391,A -85,B 0,C 180,E1 -439.351,E2 -439.351} C_VEL
LIN {X 0,Y 608.476,Z 525.856,A -85,B 0,C 180,E1 -440.527,E2 -440.527} C_VEL
LIN {X 0,Y 608.456,Z 533.731,A -85,B 0,C 180,E1 -441.699,E2 -441.699} C_VEL
LIN {X 0,Y 608.441,Z 541.089,A -85,B 0,C 180,E1 -443.034,E2 -443.034} C_VEL
LIN {X 0,Y 608.45,Z 546.925,A -85,B 0,C 180,E1 -444.366,E2 -444.366} C_VEL
LIN {X 0,Y 608.427,Z 550.384,A -85,B 0,C 180,E1 -445.362,E2 -445.362} C_VEL
LIN {X 0,Y 608.421,Z 553.886,A -85,B 0,C 180,E1 -446.689,E2 -446.689} C_VEL
LIN {X 0,Y 608.444,Z 556.192,A -85,B 0,C 180,E1 -448.014,E2 -448.014} C_VEL
LIN {X 0,Y 608.436,Z 557.351,A -85,B 0,C 180,E1 -449.338,E2 -449.338} C_VEL
LIN {X 0,Y 608.436,Z 557.35,A -85,B 0,C 180,E1 -450.662,E2 -450.662} C_VEL
LIN {X 0,Y 608.444,Z 556.191,A -85,B 0,C 180,E1 -451.986,E2 -451.986} C_VEL
LIN {X 0,Y 608.421,Z 553.885,A -85,B 0,C 180,E1 -453.311,E2 -453.311} C_VEL
LIN {X 0,Y 608.427,Z 550.382,A -85,B 0,C 180,E1 -454.638,E2 -454.638} C_VEL
LIN {X 0,Y 608.437,Z 545.606,A -85,B 0,C 180,E1 -455.967,E2 -455.967} C_VEL
LIN {X 0,Y 608.457,Z 539.424,A -85,B 0,C 180,E1 -457.3,E2 -457.3} C_VEL
LIN {X 0,Y 608.468,Z 531.652,A -85,B 0,C 180,E1 -458.636,E2 -458.636} C_VEL
LIN {X 0,Y 608.471,Z 523.368,A -85,B 0,C 180,E1 -459.809,E2 -459.809} C_VEL
LIN {X 0,Y 608.493,Z 512.646,A -85,B 0,C 180,E1 -461.064,E2 -461.064} C_VEL
LIN {X 0,Y 608.522,Z 501.271,A -85,B 0,C 180,E1 -462.168,E2 -462.168} C_VEL
LIN {X 0,Y 608.547,Z 489.85,A -85,B 0,C 180,E1 -463.1,E2 -463.1} C_VEL
LIN {X 0,Y 608.563,Z 477.442,A -85,B 0,C 180,E1 -463.95,E2 -463.95} C_VEL
LIN {X 0,Y 608.602,Z 463.853,A -85,B 0,C 180,E1 -464.718,E2 -464.718} C_VEL
LIN {X 0,Y 608.6,Z 449.784,A -85,B 0,C 180,E1 -465.36,E2 -465.36} C_VEL
LIN {X 0,Y 608.661,Z 434.555,A -85,B 0,C 180,E1 -465.895,E2 -465.895} C_VEL
LIN {X 0,Y 608.69,Z 419.96,A -85,B 0,C 180,E1 -466.271,E2 -466.271} C_VEL
LIN {X 0,Y 608.673,Z 405.359,A -85,B 0,C 180,E1 -466.517,E2 -466.517} C_VEL
LIN {X 0,Y 608.458,Z 401.681,A -85,B 0,C 180,E1 -466.586,E2 -466.586} C_VEL
LIN {X 0,Y 608.462,Z 391.671,A -85,B 0,C 180,E1 -469.571,E2 -469.571} C_VEL
LIN {X 0,Y 608.479,Z 382.331,A -85,B 0,C 180,E1 -472.405,E2 -472.405} C_VEL
LIN {X 0,Y 608.461,Z 372.99,A -85,B 0,C 180,E1 -475.301,E2 -475.301} C_VEL
LIN {X 0,Y 608.472,Z 364.818,A -85,B 0,C 180,E1 -477.891,E2 -477.891} C_VEL
LIN {X 0,Y 608.496,Z 356.645,A -85,B 0,C 180,E1 -480.544,E2 -480.544} C_VEL
LIN {X 0,Y 608.516,Z 348.472,A -85,B 0,C 180,E1 -483.271,E2 -483.271} C_VEL
LIN {X 0,Y 608.49,Z 340.149,A -85,B 0,C 180,E1 -486.09,E2 -486.09} C_VEL
LIN {X 0,Y 608.507,Z 333.075,A -85,B 0,C 180,E1 -488.585,E2 -488.585} C_VEL
LIN {X 0,Y 608.565,Z 325.719,A -85,B 0,C 180,E1 -491.353,E2 -491.353} C_VEL
LIN {X 0,Y 608.465,Z 325.318,A -85,B 0,C 180,E1 -491.673,E2 -491.673} C_VEL
LIN {X 0,Y 608.466,Z 325.32,A -85,B 0,C 180,E1 -494.265,E2 -494.265} C_VEL
LIN {X 0,Y 608.449,Z 325.322,A -85,B 0,C 180,E1 -497.04,E2 -497.04} C_VEL
LIN {X 0,Y 608.454,Z 325.317,A -85,B 0,C 180,E1 -499.697,E2 -499.697} C_VEL
LIN {X 0,Y 608.472,Z 325.315,A -85,B 0,C 180,E1 -502.254,E2 -502.254} C_VEL
LIN {X 0,Y 608.482,Z 325.316,A -85,B 0,C 180,E1 -505.091,E2 -505.091} C_VEL
LIN {X 0,Y 608.465,Z 325.321,A -85,B 0,C 180,E1 -507.906,E2 -507.906} C_VEL
LIN {X 0,Y 608.472,Z 325.315,A -85,B 0,C 180,E1 -510.221,E2 -510.221} C_VEL
LIN {X 0,Y 608.488,Z 325.314,A -85,B 0,C 180,E1 -512.792,E2 -512.792} C_VEL
LIN {X 0,Y 608.484,Z 325.314,A -85,B 0,C 180,E1 -515.847,E2 -515.847} C_VEL
LIN {X 0,Y 608.478,Z 325.317,A -85,B 0,C 180,E1 -518.309,E2 -518.309} C_VEL
LIN {X 0,Y 608.472,Z 325.317,A -85,B 0,C 180,E1 -521.285,E2 -521.285} C_VEL
LIN {X 0,Y 608.46,Z 325.316,A -85,B 0,C 180,E1 -523.906,E2 -523.906} C_VEL
LIN {X 0,Y 608.472,Z 325.315,A -85,B 0,C 180,E1 -526.644,E2 -526.644} C_VEL
LIN {X 0,Y 608.472,Z 325.318,A -85,B 0,C 180,E1 -529.35,E2 -529.35} C_VEL
LIN {X 0,Y 608.481,Z 325.317,A -85,B 0,C 180,E1 -532.033,E2 -532.033} C_VEL
LIN {X 0,Y 608.466,Z 325.316,A -85,B 0,C 180,E1 -534.698,E2 -534.698} C_VEL
LIN {X 0,Y 608.482,Z 325.313,A -85,B 0,C 180,E1 -537.352,E2 -537.352} C_VEL
LIN {X 0,Y 608.477,Z 325.318,A -85,B 0,C 180,E1 -540,E2 -540} C_VEL
LIN {X 0,Y 608.487,Z 325.316,A -85,B 0,C 180,E1 -542.648,E2 -542.648} C_VEL
LIN {X 0,Y 608.468,Z 325.315,A -85,B 0,C 180,E1 -545.302,E2 -545.302} C_VEL
LIN {X 0,Y 608.473,Z 325.315,A -85,B 0,C 180,E1 -547.967,E2 -547.967} C_VEL
LIN {X 0,Y 608.464,Z 325.316,A -85,B 0,C 180,E1 -549.455,E2 -549.455} C_VEL
LIN {X 0,Y 607.778,Z 325.403,A -85,B 0,C 180,E1 -550.008,E2 -550.008} C_VEL
LIN {X 0,Y 604.925,Z 325.759,A -85,B 0,C 180,E1 -550.905,E2 -550.905} C_VEL
LIN {X 0,Y 602.526,Z 326.059,A -85,B 0,C 180,E1 -551.627,E2 -551.627} C_VEL
LIN {X 0,Y 601.497,Z 326.187,A -85,B 0,C 180,E1 -552.183,E2 -552.183} C_VEL
LIN {X 0,Y 601.412,Z 326.194,A -85,B 0,C 180,E1 -552.372,E2 -552.372} C_VEL
LIN {X 0,Y 601.43,Z 326.195,A -85,B 0,C 180,E1 -554.897,E2 -554.897} C_VEL
LIN {X 0,Y 601.438,Z 326.192,A -85,B 0,C 180,E1 -556.986,E2 -556.986} C_VEL
LIN {X 0,Y 601.412,Z 326.197,A -85,B 0,C 180,E1 -559.809,E2 -559.809} C_VEL
LIN {X 0,Y 601.415,Z 326.2,A -85,B 0,C 180,E1 -562.683,E2 -562.683} C_VEL
LIN {X 0,Y 601.408,Z 326.194,A -85,B 0,C 180,E1 -564.878,E2 -564.878} C_VEL
LIN {X 0,Y 601.421,Z 326.197,A -85,B 0,C 180,E1 -567.363,E2 -567.363} C_VEL
LIN {X 0,Y 601.432,Z 326.196,A -85,B 0,C 180,E1 -570.164,E2 -570.164} C_VEL
LIN {X 0,Y 601.418,Z 326.193,A -85,B 0,C 180,E1 -572.714,E2 -572.714} C_VEL
LIN {X 0,Y 601.401,Z 326.198,A -85,B 0,C 180,E1 -575.112,E2 -575.112} C_VEL
LIN {X 0,Y 601.437,Z 326.192,A -85,B 0,C 180,E1 -577.419,E2 -577.419} C_VEL
LIN {X 0,Y 601.415,Z 326.194,A -85,B 0,C 180,E1 -579.995,E2 -579.995} C_VEL
LIN {X 0,Y 601.412,Z 326.198,A -85,B 0,C 180,E1 -582.67,E2 -582.67} C_VEL
LIN {X 0,Y 601.429,Z 326.198,A -85,B 0,C 180,E1 -585.482,E2 -585.482} C_VEL
LIN {X 0,Y 601.428,Z 326.196,A -85,B 0,C 180,E1 -588.407,E2 -588.407} C_VEL
LIN {X 0,Y 601.384,Z 328.092,A -85,B 0,C 180,E1 -590.471,E2 -590.471} C_VEL
LIN {X 0,Y 601.37,Z 331.146,A -85,B 0,C 180,E1 -593.414,E2 -593.414} C_VEL
LIN {X 0,Y 601.384,Z 333.933,A -85,B 0,C 180,E1 -596.071,E2 -596.071} C_VEL
LIN {X 0,Y 601.37,Z 336.593,A -85,B 0,C 180,E1 -598.553,E2 -598.553} C_VEL
LIN {X 0,Y 601.342,Z 339.975,A -85,B 0,C 180,E1 -601.368,E2 -601.368} C_VEL
LIN {X 0,Y 601.346,Z 343.401,A -85,B 0,C 180,E1 -604.146,E2 -604.146} C_VEL
LIN {X 0,Y 601.334,Z 346.478,A -85,B 0,C 180,E1 -606.586,E2 -606.586} C_VEL
LIN {X 0,Y 601.345,Z 350.195,A -85,B 0,C 180,E1 -609.475,E2 -609.475} C_VEL
LIN {X 0,Y 601.31,Z 353.912,A -85,B 0,C 180,E1 -612.309,E2 -612.309} C_VEL
LIN {X 0,Y 601.344,Z 355.326,A -85,B 0,C 180,E1 -613.32,E2 -613.32} C_VEL
LIN {X 0,Y 601.881,Z 359.388,A -85,B 0,C 180,E1 -613.394,E2 -613.394} C_VEL
LIN {X 0,Y 601.838,Z 374.124,A -85,B 0,C 180,E1 -613.683,E2 -613.683} C_VEL
LIN {X 0,Y 601.767,Z 389.153,A -85,B 0,C 180,E1 -614.114,E2 -614.114} C_VEL
LIN {X 0,Y 601.742,Z 403.761,A -85,B 0,C 180,E1 -614.678,E2 -614.678} C_VEL
LIN {X 0,Y 601.652,Z 417.846,A -85,B 0,C 180,E1 -615.368,E2 -615.368} C_VEL
LIN {X 0,Y 601.621,Z 431.769,A -85,B 0,C 180,E1 -616.215,E2 -616.215} C_VEL
LIN {X 0,Y 601.531,Z 444.726,A -85,B 0,C 180,E1 -617.174,E2 -617.174} C_VEL
LIN {X 0,Y 601.489,Z 456.278,A -85,B 0,C 180,E1 -618.201,E2 -618.201} C_VEL
LIN {X 0,Y 601.43,Z 465.993,A -85,B 0,C 180,E1 -619.224,E2 -619.224} C_VEL
LIN {X 0,Y 601.429,Z 475.524,A -85,B 0,C 180,E1 -620.414,E2 -620.414} C_VEL
LIN {X 0,Y 601.378,Z 483.459,A -85,B 0,C 180,E1 -621.6,E2 -621.6} C_VEL
LIN {X 0,Y 601.368,Z 490.87,A -85,B 0,C 180,E1 -622.951,E2 -622.951} C_VEL
LIN {X 0,Y 601.373,Z 496.758,A -85,B 0,C 180,E1 -624.299,E2 -624.299} C_VEL
LIN {X 0,Y 601.327,Z 500.24,A -85,B 0,C 180,E1 -625.307,E2 -625.307} C_VEL
LIN {X 0,Y 601.336,Z 503.789,A -85,B 0,C 180,E1 -626.65,E2 -626.65} C_VEL
LIN {X 0,Y 601.343,Z 506.139,A -85,B 0,C 180,E1 -627.99,E2 -627.99} C_VEL
LIN {X 0,Y 601.334,Z 507.337,A -85,B 0,C 180,E1 -629.33,E2 -629.33} C_VEL
LIN {X 0,Y 601.335,Z 507.361,A -85,B 0,C 180,E1 -630.669,E2 -630.669} C_VEL
LIN {X 0,Y 601.343,Z 506.245,A -85,B 0,C 180,E1 -632.009,E2 -632.009} C_VEL
LIN {X 0,Y 601.339,Z 503.983,A -85,B 0,C 180,E1 -633.35,E2 -633.35} C_VEL
LIN {X 0,Y 601.328,Z 500.526,A -85,B 0,C 180,E1 -634.692,E2 -634.692} C_VEL
LIN {X 0,Y 601.358,Z 495.799,A -85,B 0,C 180,E1 -636.037,E2 -636.037} C_VEL
LIN {X 0,Y 601.365,Z 489.668,A -85,B 0,C 180,E1 -637.386,E2 -637.386} C_VEL
LIN {X 0,Y 601.389,Z 481.952,A -85,B 0,C 180,E1 -638.738,E2 -638.738} C_VEL
LIN {X 0,Y 601.428,Z 473.709,A -85,B 0,C 180,E1 -639.925,E2 -639.925} C_VEL
LIN {X 0,Y 601.443,Z 463.367,A -85,B 0,C 180,E1 -641.164,E2 -641.164} C_VEL
LIN {X 0,Y 601.503,Z 451.788,A -85,B 0,C 180,E1 -642.312,E2 -642.312} C_VEL
LIN {X 0,Y 601.557,Z 440.466,A -85,B 0,C 180,E1 -643.254,E2 -643.254} C_VEL
LIN {X 0,Y 601.623,Z 427.318,A -85,B 0,C 180,E1 -644.167,E2 -644.167} C_VEL
LIN {X 0,Y 601.673,Z 414.764,A -85,B 0,C 180,E1 -644.89,E2 -644.89} C_VEL
LIN {X 0,Y 601.731,Z 399.841,A -85,B 0,C 180,E1 -645.583,E2 -645.583} C_VEL
LIN {X 0,Y 601.816,Z 385.355,A -85,B 0,C 180,E1 -646.102,E2 -646.102} C_VEL
LIN {X 0,Y 601.866,Z 370.103,A -85,B 0,C 180,E1 -646.502,E2 -646.502} C_VEL
LIN {X 0,Y 601.76,Z 357.435,A -85,B 0,C 180,E1 -646.727,E2 -646.727} C_VEL
LIN {X 0,Y 601.338,Z 355.235,A -85,B 0,C 180,E1 -646.782,E2 -646.782} C_VEL
LIN {X 0,Y 601.313,Z 352.172,A -85,B 0,C 180,E1 -649.102,E2 -649.102} C_VEL
LIN {X 0,Y 601.315,Z 349.383,A -85,B 0,C 180,E1 -651.242,E2 -651.242} C_VEL
LIN {X 0,Y 601.342,Z 345.664,A -85,B 0,C 180,E1 -654.145,E2 -654.145} C_VEL
LIN {X 0,Y 601.34,Z 342.875,A -85,B 0,C 180,E1 -656.366,E2 -656.366} C_VEL
LIN {X 0,Y 601.341,Z 339.155,A -85,B 0,C 180,E1 -659.397,E2 -659.397} C_VEL
LIN {X 0,Y 601.339,Z 336.372,A -85,B 0,C 180,E1 -661.73,E2 -661.73} C_VEL
LIN {X 0,Y 601.381,Z 333.831,A -85,B 0,C 180,E1 -664.121,E2 -664.121} C_VEL
LIN {X 0,Y 601.367,Z 331.24,A -85,B 0,C 180,E1 -666.585,E2 -666.585} C_VEL
LIN {X 0,Y 601.384,Z 328.614,A -85,B 0,C 180,E1 -669.128,E2 -669.128} C_VEL
LIN {X 0,Y 601.396,Z 326.201,A -85,B 0,C 180,E1 -671.59,E2 -671.59} C_VEL
LIN {X 0,Y 601.449,Z 326.19,A -85,B 0,C 180,E1 -673.584,E2 -673.584} C_VEL
LIN {X 0,Y 601.428,Z 326.194,A -85,B 0,C 180,E1 -676.427,E2 -676.427} C_VEL
LIN {X 0,Y 601.413,Z 326.2,A -85,B 0,C 180,E1 -679.125,E2 -679.125} C_VEL
LIN {X 0,Y 601.421,Z 326.194,A -85,B 0,C 180,E1 -681.732,E2 -681.732} C_VEL
LIN {X 0,Y 601.408,Z 326.195,A -85,B 0,C 180,E1 -684.247,E2 -684.247} C_VEL
LIN {X 0,Y 601.417,Z 326.199,A -85,B 0,C 180,E1 -686.686,E2 -686.686} C_VEL
LIN {X 0,Y 601.433,Z 326.191,A -85,B 0,C 180,E1 -689.059,E2 -689.059} C_VEL
LIN {X 0,Y 601.431,Z 326.197,A -85,B 0,C 180,E1 -691.373,E2 -691.373} C_VEL
LIN {X 0,Y 601.405,Z 326.194,A -85,B 0,C 180,E1 -693.636,E2 -693.636} C_VEL
LIN {X 0,Y 601.421,Z 326.193,A -85,B 0,C 180,E1 -696.59,E2 -696.59} C_VEL
LIN {X 0,Y 601.427,Z 326.191,A -85,B 0,C 180,E1 -699.478,E2 -699.478} C_VEL
LIN {X 0,Y 601.402,Z 326.197,A -85,B 0,C 180,E1 -702.312,E2 -702.312} C_VEL
LIN {X 0,Y 601.416,Z 326.193,A -85,B 0,C 180,E1 -704.409,E2 -704.409} C_VEL
LIN {X 0,Y 601.421,Z 326.192,A -85,B 0,C 180,E1 -707.172,E2 -707.172} C_VEL
LIN {X 0,Y 601.43,Z 326.194,A -85,B 0,C 180,E1 -709.905,E2 -709.905} C_VEL
LIN {X 0,Y 601.439,Z 326.197,A -85,B 0,C 180,E1 -712.615,E2 -712.615} C_VEL
LIN {X 0,Y 601.421,Z 326.195,A -85,B 0,C 180,E1 -715.308,E2 -715.308} C_VEL
LIN {X 0,Y 601.419,Z 326.193,A -85,B 0,C 180,E1 -717.991,E2 -717.991} C_VEL
LIN {X 0,Y 601.45,Z 326.19,A -85,B 0,C 180,E1 -720.669,E2 -720.669} C_VEL
LIN {X 0,Y 601.435,Z 326.196,A -85,B 0,C 180,E1 -723.349,E2 -723.349} C_VEL
LIN {X 0,Y 601.407,Z 326.197,A -85,B 0,C 180,E1 -726.037,E2 -726.037} C_VEL
LIN {X 0,Y 601.414,Z 326.194,A -85,B 0,C 180,E1 -728.738,E2 -728.738} C_VEL
LIN {X 0,Y 601.435,Z 326.191,A -85,B 0,C 180,E1 -731.458,E2 -731.458} C_VEL
LIN {X 0,Y 601.418,Z 326.196,A -85,B 0,C 180,E1 -734.205,E2 -734.205} C_VEL
LIN {X 0,Y 601.433,Z 326.197,A -85,B 0,C 180,E1 -736.986,E2 -736.986} C_VEL
LIN {X 0,Y 601.408,Z 326.198,A -85,B 0,C 180,E1 -739.809,E2 -739.809} C_VEL
LIN {X 0,Y 601.41,Z 326.196,A -85,B 0,C 180,E1 -742.683,E2 -742.683} C_VEL
LIN {X 0,Y 601.405,Z 326.197,A -85,B 0,C 180,E1 -744.878,E2 -744.878} C_VEL
LIN {X 0,Y 601.422,Z 326.196,A -85,B 0,C 180,E1 -747.867,E2 -747.867} C_VEL
LIN {X 0,Y 601.447,Z 326.19,A -85,B 0,C 180,E1 -750.163,E2 -750.163} C_VEL
LIN {X 0,Y 601.416,Z 326.194,A -85,B 0,C 180,E1 -752.715,E2 -752.715} C_VEL
LIN {X 0,Y 601.414,Z 326.198,A -85,B 0,C 180,E1 -755.115,E2 -755.115} C_VEL
LIN {X 0,Y 601.434,Z 326.191,A -85,B 0,C 180,E1 -757.419,E2 -757.419} C_VEL
LIN {X 0,Y 601.409,Z 326.198,A -85,B 0,C 180,E1 -759.995,E2 -759.995} C_VEL
LIN {X 0,Y 601.408,Z 326.199,A -85,B 0,C 180,E1 -762.671,E2 -762.671} C_VEL
LIN {X 0,Y 601.424,Z 326.194,A -85,B 0,C 180,E1 -765.482,E2 -765.482} C_VEL
LIN {X 0,Y 601.44,Z 326.303,A -85,B 0,C 180,E1 -768.293,E2 -768.293} C_VEL
LIN {X 0,Y 601.557,Z 330.662,A -85,B 0,C 180,E1 -770.017,E2 -770.017} C_VEL
LIN {X 0,Y 601.536,Z 337.743,A -85,B 0,C 180,E1 -772.605,E2 -772.605} C_VEL
LIN {X 0,Y 601.528,Z 345.985,A -85,B 0,C 180,E1 -775.483,E2 -775.483} C_VEL
LIN {X 0,Y 601.526,Z 354.312,A -85,B 0,C 180,E1 -778.281,E2 -778.281} C_VEL
LIN {X 0,Y 601.496,Z 363.114,A -85,B 0,C 180,E1 -781.201,E2 -781.201} C_VEL
LIN {X 0,Y 601.435,Z 372.193,A -85,B 0,C 180,E1 -784.128,E2 -784.128} C_VEL
LIN {X 0,Y 601.431,Z 381.165,A -85,B 0,C 180,E1 -786.955,E2 -786.955} C_VEL
LIN {X 0,Y 601.423,Z 390.505,A -85,B 0,C 180,E1 -789.835,E2 -789.835} C_VEL
LIN {X 0,Y 601.389,Z 399.845,A -85,B 0,C 180,E1 -792.663,E2 -792.663} C_VEL
LIN {X 0,Y 601.388,Z 401.767,A -85,B 0,C 180,E1 -793.231,E2 -793.231} C_VEL
LIN {X 0,Y 601.864,Z 405.64,A -85,B 0,C 180,E1 -793.295,E2 -793.295} C_VEL
LIN {X 0,Y 601.855,Z 420.757,A -85,B 0,C 180,E1 -793.558,E2 -793.558} C_VEL
LIN {X 0,Y 601.807,Z 435.308,A -85,B 0,C 180,E1 -793.941,E2 -793.941} C_VEL
LIN {X 0,Y 601.737,Z 449.8,A -85,B 0,C 180,E1 -794.461,E2 -794.461} C_VEL
LIN {X 0,Y 601.691,Z 463.868,A -85,B 0,C 180,E1 -795.11,E2 -795.11} C_VEL
LIN {X 0,Y 601.613,Z 477.589,A -85,B 0,C 180,E1 -795.894,E2 -795.894} C_VEL
LIN {X 0,Y 601.57,Z 491.018,A -85,B 0,C 180,E1 -796.832,E2 -796.832} C_VEL
LIN {X 0,Y 601.513,Z 503.195,A -85,B 0,C 180,E1 -797.86,E2 -797.86} C_VEL
LIN {X 0,Y 601.437,Z 514.273,A -85,B 0,C 180,E1 -798.982,E2 -798.982} C_VEL
LIN {X 0,Y 601.427,Z 523.372,A -85,B 0,C 180,E1 -800.075,E2 -800.075} C_VEL
LIN {X 0,Y 601.388,Z 531.656,A -85,B 0,C 180,E1 -801.262,E2 -801.262} C_VEL
LIN {X 0,Y 601.365,Z 539.427,A -85,B 0,C 180,E1 -802.614,E2 -802.614} C_VEL
LIN {X 0,Y 601.357,Z 545.609,A -85,B 0,C 180,E1 -803.963,E2 -803.963} C_VEL
LIN {X 0,Y 601.33,Z 550.384,A -85,B 0,C 180,E1 -805.308,E2 -805.308} C_VEL
LIN {X 0,Y 601.337,Z 553.887,A -85,B 0,C 180,E1 -806.65,E2 -806.65} C_VEL
LIN {X 0,Y 601.343,Z 556.192,A -85,B 0,C 180,E1 -807.991,E2 -807.991} C_VEL
LIN {X 0,Y 601.337,Z 557.35,A -85,B 0,C 180,E1 -809.331,E2 -809.331} C_VEL
LIN {X 0,Y 601.337,Z 557.35,A -85,B 0,C 180,E1 -810.67,E2 -810.67} C_VEL
LIN {X 0,Y 601.343,Z 556.191,A -85,B 0,C 180,E1 -812.01,E2 -812.01} C_VEL
LIN {X 0,Y 601.337,Z 553.885,A -85,B 0,C 180,E1 -813.35,E2 -813.35} C_VEL
LIN {X 0,Y 601.33,Z 550.382,A -85,B 0,C 180,E1 -814.693,E2 -814.693} C_VEL
LIN {X 0,Y 601.357,Z 545.607,A -85,B 0,C 180,E1 -816.038,E2 -816.038} C_VEL
LIN {X 0,Y 601.366,Z 539.424,A -85,B 0,C 180,E1 -817.386,E2 -817.386} C_VEL
LIN {X 0,Y 601.389,Z 531.651,A -85,B 0,C 180,E1 -818.739,E2 -818.739} C_VEL
LIN {X 0,Y 601.427,Z 523.368,A -85,B 0,C 180,E1 -819.925,E2 -819.925} C_VEL
LIN {X 0,Y 601.461,Z 512.927,A -85,B 0,C 180,E1 -821.165,E2 -821.165} C_VEL
LIN {X 0,Y 601.514,Z 503.189,A -85,B 0,C 180,E1 -822.141,E2 -822.141} C_VEL
LIN {X 0,Y 601.57,Z 491.011,A -85,B 0,C 180,E1 -823.169,E2 -823.169} C_VEL
LIN {X 0,Y 601.607,Z 479.073,A -85,B 0,C 180,E1 -824.012,E2 -824.012} C_VEL
LIN {X 0,Y 601.674,Z 465.522,A -85,B 0,C 180,E1 -824.804,E2 -824.804} C_VEL
LIN {X 0,Y 601.724,Z 450.837,A -85,B 0,C 180,E1 -825.496,E2 -825.496} C_VEL
LIN {X 0,Y 601.793,Z 436.609,A -85,B 0,C 180,E1 -826.016,E2 -826.016} C_VEL
LIN {X 0,Y 601.851,Z 421.623,A -85,B 0,C 180,E1 -826.422,E2 -826.422} C_VEL
LIN {X 0,Y 601.865,Z 406.279,A -85,B 0,C 180,E1 -826.696,E2 -826.696} C_VEL
LIN {X 0,Y 601.39,Z 401.763,A -85,B 0,C 180,E1 -826.769,E2 -826.769} C_VEL
LIN {X 0,Y 601.425,Z 392.838,A -85,B 0,C 180,E1 -829.454,E2 -829.454} C_VEL
LIN {X 0,Y 601.432,Z 383.622,A -85,B 0,C 180,E1 -832.282,E2 -832.282} C_VEL
LIN {X 0,Y 601.449,Z 374.158,A -85,B 0,C 180,E1 -835.246,E2 -835.246} C_VEL
LIN {X 0,Y 601.451,Z 365.985,A -85,B 0,C 180,E1 -837.866,E2 -837.866} C_VEL
LIN {X 0,Y 601.492,Z 357.813,A -85,B 0,C 180,E1 -840.549,E2 -840.549} C_VEL
LIN {X 0,Y 601.526,Z 349.6,A -85,B 0,C 180,E1 -843.308,E2 -843.308} C_VEL
LIN {X 0,Y 601.537,Z 342.417,A -85,B 0,C 180,E1 -845.745,E2 -845.745} C_VEL
LIN {X 0,Y 601.523,Z 334.697,A -85,B 0,C 180,E1 -848.482,E2 -848.482} C_VEL
LIN {X 0,Y 601.596,Z 328.402,A -85,B 0,C 180,E1 -850.86,E2 -850.86} C_VEL
LIN {X 0,Y 601.431,Z 326.196,A -85,B 0,C 180,E1 -851.765,E2 -851.765} C_VEL
LIN {X 0,Y 601.427,Z 326.194,A -85,B 0,C 180,E1 -854.535,E2 -854.535} C_VEL
LIN {X 0,Y 601.41,Z 326.197,A -85,B 0,C 180,E1 -857.41,E2 -857.41} C_VEL
LIN {X 0,Y 601.405,Z 326.198,A -85,B 0,C 180,E1 -860.005,E2 -860.005} C_VEL
LIN {X 0,Y 601.437,Z 326.191,A -85,B 0,C 180,E1 -862.618,E2 -862.618} C_VEL
LIN {X 0,Y 601.439,Z 326.193,A -85,B 0,C 180,E1 -865.07,E2 -865.07} C_VEL
LIN {X 0,Y 601.427,Z 326.194,A -85,B 0,C 180,E1 -867.484,E2 -867.484} C_VEL
LIN {X 0,Y 601.432,Z 326.192,A -85,B 0,C 180,E1 -869.852,E2 -869.852} C_VEL
LIN {X 0,Y 601.425,Z 326.195,A -85,B 0,C 180,E1 -872.636,E2 -872.636} C_VEL
LIN {X 0,Y 601.407,Z 326.197,A -85,B 0,C 180,E1 -875.122,E2 -875.122} C_VEL
LIN {X 0,Y 601.418,Z 326.194,A -85,B 0,C 180,E1 -877.395,E2 -877.395} C_VEL
LIN {X 0,Y 601.408,Z 326.198,A -85,B 0,C 180,E1 -880.191,E2 -880.191} C_VEL
LIN {X 0,Y 601.435,Z 326.197,A -85,B 0,C 180,E1 -883.014,E2 -883.014} C_VEL
LIN {X 0,Y 601.425,Z 326.196,A -85,B 0,C 180,E1 -885.908,E2 -885.908} C_VEL
LIN {X 0,Y 601.438,Z 326.191,A -85,B 0,C 180,E1 -888.542,E2 -888.542} C_VEL
LIN {X 0,Y 601.416,Z 326.194,A -85,B 0,C 180,E1 -891.262,E2 -891.262} C_VEL
LIN {X 0,Y 601.409,Z 326.197,A -85,B 0,C 180,E1 -893.963,E2 -893.963} C_VEL
LIN {X 0,Y 601.437,Z 326.195,A -85,B 0,C 180,E1 -896.651,E2 -896.651} C_VEL
LIN {X 0,Y 601.451,Z 326.19,A -85,B 0,C 180,E1 -899.331,E2 -899.331} C_VEL
LIN {X 0,Y 601.42,Z 326.193,A -85,B 0,C 180,E1 -902.009,E2 -902.009} C_VEL
LIN {X 0,Y 601.425,Z 326.195,A -85,B 0,C 180,E1 -904.692,E2 -904.692} C_VEL
LIN {X 0,Y 601.442,Z 326.196,A -85,B 0,C 180,E1 -907.385,E2 -907.385} C_VEL
LIN {X 0,Y 601.431,Z 326.193,A -85,B 0,C 180,E1 -910.095,E2 -910.095} C_VEL
LIN {X 0,Y 601.412,Z 326.194,A -85,B 0,C 180,E1 -912.372,E2 -912.372} C_VEL
LIN {X 0,Y 600.745,Z 326.276,A -85,B 0,C 180,E1 -912.931,E2 -912.931} C_VEL
LIN {X 0,Y 597.895,Z 326.635,A -85,B 0,C 180,E1 -913.839,E2 -913.839} C_VEL
LIN {X 0,Y 595.486,Z 326.938,A -85,B 0,C 180,E1 -914.569,E2 -914.569} C_VEL
LIN {X 0,Y 594.449,Z 327.066,A -85,B 0,C 180,E1 -915.133,E2 -915.133} C_VEL
LIN {X 0,Y 594.363,Z 327.074,A -85,B 0,C 180,E1 -915.323,E2 -915.323} C_VEL
LIN {X 0,Y 594.381,Z 327.073,A -85,B 0,C 180,E1 -917.904,E2 -917.904} C_VEL
LIN {X 0,Y 594.375,Z 327.072,A -85,B 0,C 180,E1 -920.915,E2 -920.915} C_VEL
LIN {X 0,Y 594.381,Z 327.07,A -85,B 0,C 180,E1 -923.705,E2 -923.705} C_VEL
LIN {X 0,Y 594.392,Z 327.07,A -85,B 0,C 180,E1 -926.023,E2 -926.023} C_VEL
LIN {X 0,Y 594.386,Z 327.073,A -85,B 0,C 180,E1 -928.958,E2 -928.958} C_VEL
LIN {X 0,Y 594.386,Z 327.073,A -85,B 0,C 180,E1 -931.643,E2 -931.643} C_VEL
LIN {X 0,Y 594.386,Z 327.071,A -85,B 0,C 180,E1 -934.58,E2 -934.58} C_VEL
LIN {X 0,Y 594.388,Z 327.069,A -85,B 0,C 180,E1 -937.087,E2 -937.087} C_VEL
LIN {X 0,Y 594.38,Z 327.072,A -85,B 0,C 180,E1 -939.774,E2 -939.774} C_VEL
LIN {X 0,Y 594.37,Z 327.076,A -85,B 0,C 180,E1 -942.375,E2 -942.375} C_VEL
LIN {X 0,Y 594.367,Z 327.074,A -85,B 0,C 180,E1 -945.191,E2 -945.191} C_VEL
LIN {X 0,Y 594.385,Z 327.071,A -85,B 0,C 180,E1 -948.152,E2 -948.152} C_VEL
LIN {X 0,Y 594.322,Z 327.719,A -85,B 0,C 180,E1 -949.429,E2 -949.429} C_VEL
LIN {X 0,Y 594.325,Z 330.788,A -85,B 0,C 180,E1 -952.4,E2 -952.4} C_VEL
LIN {X 0,Y 594.32,Z 333.114,A -85,B 0,C 180,E1 -954.681,E2 -954.681} C_VEL
LIN {X 0,Y 594.298,Z 335.66,A -85,B 0,C 180,E1 -957.101,E2 -957.101} C_VEL
LIN {X 0,Y 594.272,Z 338.422,A -85,B 0,C 180,E1 -959.691,E2 -959.691} C_VEL
LIN {X 0,Y 594.264,Z 341.834,A -85,B 0,C 180,E1 -962.533,E2 -962.533} C_VEL
LIN {X 0,Y 594.278,Z 345.602,A -85,B 0,C 180,E1 -965.59,E2 -965.59} C_VEL
LIN {X 0,Y 594.222,Z 349.267,A -85,B 0,C 180,E1 -968.491,E2 -968.491} C_VEL
LIN {X 0,Y 594.24,Z 352.638,A -85,B 0,C 180,E1 -971.112,E2 -971.112} C_VEL
LIN {X 0,Y 594.264,Z 355.31,A -85,B 0,C 180,E1 -973.115,E2 -973.115} C_VEL
LIN {X 0,Y 595.1,Z 359.426,A -85,B 0,C 180,E1 -973.2,E2 -973.2} C_VEL
LIN {X 0,Y 595.015,Z 374.737,A -85,B 0,C 180,E1 -973.504,E2 -973.504} C_VEL
LIN {X 0,Y 594.93,Z 389.172,A -85,B 0,C 180,E1 -973.926,E2 -973.926} C_VEL
LIN {X 0,Y 594.866,Z 403.776,A -85,B 0,C 180,E1 -974.496,E2 -974.496} C_VEL
LIN {X 0,Y 594.761,Z 417.858,A -85,B 0,C 180,E1 -975.195,E2 -975.195} C_VEL
LIN {X 0,Y 594.676,Z 430.627,A -85,B 0,C 180,E1 -975.972,E2 -975.972} C_VEL
LIN {X 0,Y 594.555,Z 442.614,A -85,B 0,C 180,E1 -976.847,E2 -976.847} C_VEL
LIN {X 0,Y 594.49,Z 454.508,A -85,B 0,C 180,E1 -977.887,E2 -977.887} C_VEL
LIN {X 0,Y 594.439,Z 464.339,A -85,B 0,C 180,E1 -978.903,E2 -978.903} C_VEL
LIN {X 0,Y 594.369,Z 474.291,A -85,B 0,C 180,E1 -980.127,E2 -980.127} C_VEL
LIN {X 0,Y 594.342,Z 482.45,A -85,B 0,C 180,E1 -981.328,E2 -981.328} C_VEL
LIN {X 0,Y 594.287,Z 489.185,A -85,B 0,C 180,E1 -982.525,E2 -982.525} C_VEL
LIN {X 0,Y 594.279,Z 495.419,A -85,B 0,C 180,E1 -983.89,E2 -983.89} C_VEL
LIN {X 0,Y 594.23,Z 500.243,A -85,B 0,C 180,E1 -985.251,E2 -985.251} C_VEL
LIN {X 0,Y 594.256,Z 503.79,A -85,B 0,C 180,E1 -986.61,E2 -986.61} C_VEL
LIN {X 0,Y 594.241,Z 506.14,A -85,B 0,C 180,E1 -987.966,E2 -987.966} C_VEL
LIN {X 0,Y 594.235,Z 507.337,A -85,B 0,C 180,E1 -989.322,E2 -989.322} C_VEL
LIN {X 0,Y 594.236,Z 507.361,A -85,B 0,C 180,E1 -990.677,E2 -990.677} C_VEL
LIN {X 0,Y 594.242,Z 506.245,A -85,B 0,C 180,E1 -992.033,E2 -992.033} C_VEL
LIN {X 0,Y 594.258,Z 503.983,A -85,B 0,C 180,E1 -993.39,E2 -993.39} C_VEL
LIN {X 0,Y 594.231,Z 500.525,A -85,B 0,C 180,E1 -994.749,E2 -994.749} C_VEL
LIN {X 0,Y 594.279,Z 495.796,A -85,B 0,C 180,E1 -996.11,E2 -996.11} C_VEL
LIN {X 0,Y 594.287,Z 489.665,A -85,B 0,C 180,E1 -997.474,E2 -997.474} C_VEL
LIN {X 0,Y 594.332,Z 481.948,A -85,B 0,C 180,E1 -998.843,E2 -998.843} C_VEL
LIN {X 0,Y 594.387,Z 473.706,A -85,B 0,C 180,E1 -1000.044,E2 -1000.044} C_VEL
LIN {X 0,Y 594.41,Z 463.981,A -85,B 0,C 180,E1 -1001.229,E2 -1001.229} C_VEL
LIN {X 0,Y 594.516,Z 453.658,A -85,B 0,C 180,E1 -1002.285,E2 -1002.285} C_VEL
LIN {X 0,Y 594.578,Z 441.588,A -85,B 0,C 180,E1 -1003.326,E2 -1003.326} C_VEL
LIN {X 0,Y 594.683,Z 428.14,A -85,B 0,C 180,E1 -1004.285,E2 -1004.285} C_VEL
LIN {X 0,Y 594.781,Z 414.754,A -85,B 0,C 180,E1 -1005.067,E2 -1005.067} C_VEL
LIN {X 0,Y 594.885,Z 399.828,A -85,B 0,C 180,E1 -1005.767,E2 -1005.767} C_VEL
LIN {X 0,Y 594.997,Z 385.337,A -85,B 0,C 180,E1 -1006.292,E2 -1006.292} C_VEL
LIN {X 0,Y 595.065,Z 370.039,A -85,B 0,C 180,E1 -1006.697,E2 -1006.697} C_VEL
LIN {X 0,Y 594.971,Z 358.843,A -85,B 0,C 180,E1 -1006.903,E2 -1006.903} C_VEL
LIN {X 0,Y 594.249,Z 355.246,A -85,B 0,C 180,E1 -1006.979,E2 -1006.979} C_VEL
LIN {X 0,Y 594.238,Z 352.172,A -85,B 0,C 180,E1 -1009.338,E2 -1009.338} C_VEL
LIN {X 0,Y 594.221,Z 349.382,A -85,B 0,C 180,E1 -1011.508,E2 -1011.508} C_VEL
LIN {X 0,Y 594.274,Z 345.663,A -85,B 0,C 180,E1 -1014.451,E2 -1014.451} C_VEL
LIN {X 0,Y 594.257,Z 342.874,A -85,B 0,C 180,E1 -1016.705,E2 -1016.705} C_VEL
LIN {X 0,Y 594.255,Z 340.084,A -85,B 0,C 180,E1 -1019.005,E2 -1019.005} C_VEL
LIN {X 0,Y 594.294,Z 337.078,A -85,B 0,C 180,E1 -1021.629,E2 -1021.629} C_VEL
LIN {X 0,Y 594.308,Z 333.998,A -85,B 0,C 180,E1 -1024.584,E2 -1024.584} C_VEL
LIN {X 0,Y 594.322,Z 331.402,A -85,B 0,C 180,E1 -1027.091,E2 -1027.091} C_VEL
LIN {X 0,Y 594.314,Z 328.639,A -85,B 0,C 180,E1 -1029.767,E2 -1029.767} C_VEL
LIN {X 0,Y 594.355,Z 327.079,A -85,B 0,C 180,E1 -1031.466,E2 -1031.466} C_VEL
LIN {X 0,Y 594.381,Z 327.072,A -85,B 0,C 180,E1 -1034.236,E2 -1034.236} C_VEL
LIN {X 0,Y 594.363,Z 327.073,A -85,B 0,C 180,E1 -1037.148,E2 -1037.148} C_VEL
LIN {X 0,Y 594.367,Z 327.074,A -85,B 0,C 180,E1 -1039.433,E2 -1039.433} C_VEL
LIN {X 0,Y 594.389,Z 327.072,A -85,B 0,C 180,E1 -1042.391,E2 -1042.391} C_VEL
LIN {X 0,Y 594.385,Z 327.07,A -85,B 0,C 180,E1 -1044.671,E2 -1044.671} C_VEL
LIN {X 0,Y 594.375,Z 327.072,A -85,B 0,C 180,E1 -1047.088,E2 -1047.088} C_VEL
LIN {X 0,Y 594.401,Z 327.072,A -85,B 0,C 180,E1 -1049.669,E2 -1049.669} C_VEL
LIN {X 0,Y 594.373,Z 327.072,A -85,B 0,C 180,E1 -1052.539,E2 -1052.539} C_VEL
LIN {X 0,Y 594.382,Z 327.071,A -85,B 0,C 180,E1 -1054.807,E2 -1054.807} C_VEL
LIN {X 0,Y 594.365,Z 327.076,A -85,B 0,C 180,E1 -1057.264,E2 -1057.264} C_VEL
LIN {X 0,Y 594.377,Z 327.069,A -85,B 0,C 180,E1 -1059.946,E2 -1059.946} C_VEL
LIN {X 0,Y 594.393,Z 327.068,A -85,B 0,C 180,E1 -1062.807,E2 -1062.807} C_VEL
LIN {X 0,Y 594.387,Z 327.068,A -85,B 0,C 180,E1 -1065.826,E2 -1065.826} C_VEL
LIN {X 0,Y 594.395,Z 327.069,A -85,B 0,C 180,E1 -1068.404,E2 -1068.404} C_VEL
LIN {X 0,Y 594.401,Z 327.073,A -85,B 0,C 180,E1 -1071.158,E2 -1071.158} C_VEL
LIN {X 0,Y 594.377,Z 327.073,A -85,B 0,C 180,E1 -1073.891,E2 -1073.891} C_VEL
LIN {X 0,Y 594.384,Z 327.07,A -85,B 0,C 180,E1 -1076.611,E2 -1076.611} C_VEL
LIN {X 0,Y 594.421,Z 327.065,A -85,B 0,C 180,E1 -1079.322,E2 -1079.322} C_VEL
LIN {X 0,Y 594.396,Z 327.07,A -85,B 0,C 180,E1 -1082.033,E2 -1082.033} C_VEL
LIN {X 0,Y 594.4,Z 327.073,A -85,B 0,C 180,E1 -1084.747,E2 -1084.747} C_VEL
LIN {X 0,Y 594.394,Z 327.07,A -85,B 0,C 180,E1 -1087.473,E2 -1087.473} C_VEL
LIN {X 0,Y 594.392,Z 327.068,A -85,B 0,C 180,E1 -1090.216,E2 -1090.216} C_VEL
LIN {X 0,Y 594.37,Z 327.071,A -85,B 0,C 180,E1 -1092.983,E2 -1092.983} C_VEL
LIN {X 0,Y 594.369,Z 327.073,A -85,B 0,C 180,E1 -1095.781,E2 -1095.781} C_VEL
LIN {X 0,Y 594.385,Z 327.074,A -85,B 0,C 180,E1 -1098.617,E2 -1098.617} C_VEL
LIN {X 0,Y 594.37,Z 327.077,A -85,B 0,C 180,E1 -1101.503,E2 -1101.503} C_VEL
LIN {X 0,Y 594.388,Z 327.073,A -85,B 0,C 180,E1 -1104.446,E2 -1104.446} C_VEL
LIN {X 0,Y 594.39,Z 327.073,A -85,B 0,C 180,E1 -1107.46,E2 -1107.46} C_VEL
LIN {X 0,Y 594.4,Z 327.07,A -85,B 0,C 180,E1 -1110.331,E2 -1110.331} C_VEL
LIN {X 0,Y 594.375,Z 327.071,A -85,B 0,C 180,E1 -1112.95,E2 -1112.95} C_VEL
LIN {X 0,Y 594.382,Z 327.074,A -85,B 0,C 180,E1 -1115.407,E2 -1115.407} C_VEL
LIN {X 0,Y 594.39,Z 327.071,A -85,B 0,C 180,E1 -1117.94,E2 -1117.94} C_VEL
LIN {X 0,Y 594.381,Z 327.071,A -85,B 0,C 180,E1 -1120.823,E2 -1120.823} C_VEL
LIN {X 0,Y 594.366,Z 327.073,A -85,B 0,C 180,E1 -1123.84,E2 -1123.84} C_VEL
LIN {X 0,Y 594.38,Z 327.072,A -85,B 0,C 180,E1 -1126.702,E2 -1126.702} C_VEL
LIN {X 0,Y 594.395,Z 327.198,A -85,B 0,C 180,E1 -1128.063,E2 -1128.063} C_VEL
LIN {X 0,Y 594.638,Z 330.601,A -85,B 0,C 180,E1 -1129.456,E2 -1129.456} C_VEL
LIN {X 0,Y 594.565,Z 338.411,A -85,B 0,C 180,E1 -1132.37,E2 -1132.37} C_VEL
LIN {X 0,Y 594.521,Z 345.932,A -85,B 0,C 180,E1 -1135.043,E2 -1135.043} C_VEL
LIN {X 0,Y 594.538,Z 354.26,A -85,B 0,C 180,E1 -1137.864,E2 -1137.864} C_VEL
LIN {X 0,Y 594.497,Z 362.485,A -85,B 0,C 180,E1 -1140.62,E2 -1140.62} C_VEL
LIN {X 0,Y 594.444,Z 371.806,A -85,B 0,C 180,E1 -1143.676,E2 -1143.676} C_VEL
LIN {X 0,Y 594.405,Z 381.165,A -85,B 0,C 180,E1 -1146.666,E2 -1146.666} C_VEL
LIN {X 0,Y 594.382,Z 390.505,A -85,B 0,C 180,E1 -1149.586,E2 -1149.586} C_VEL
LIN {X 0,Y 594.328,Z 399.845,A -85,B 0,C 180,E1 -1152.45,E2 -1152.45} C_VEL
LIN {X 0,Y 594.32,Z 401.717,A -85,B 0,C 180,E1 -1153.019,E2 -1153.019} C_VEL
LIN {X 0,Y 595.079,Z 405.933,A -85,B 0,C 180,E1 -1153.103,E2 -1153.103} C_VEL
LIN {X 0,Y 595.056,Z 421.297,A -85,B 0,C 180,E1 -1153.378,E2 -1153.378} C_VEL
LIN {X 0,Y 594.99,Z 435.307,A -85,B 0,C 180,E1 -1153.752,E2 -1153.752} C_VEL
LIN {X 0,Y 594.867,Z 449.802,A -85,B 0,C 180,E1 -1154.277,E2 -1154.277} C_VEL
LIN {X 0,Y 594.796,Z 463.871,A -85,B 0,C 180,E1 -1154.933,E2 -1154.933} C_VEL
LIN {X 0,Y 594.682,Z 477.412,A -85,B 0,C 180,E1 -1155.715,E2 -1155.715} C_VEL
LIN {X 0,Y 594.587,Z 489.86,A -85,B 0,C 180,E1 -1156.587,E2 -1156.587} C_VEL
LIN {X 0,Y 594.535,Z 501.279,A -85,B 0,C 180,E1 -1157.542,E2 -1157.542} C_VEL
LIN {X 0,Y 594.434,Z 511.712,A -85,B 0,C 180,E1 -1158.572,E2 -1158.572} C_VEL
LIN {X 0,Y 594.38,Z 522.023,A -85,B 0,C 180,E1 -1159.784,E2 -1159.784} C_VEL
LIN {X 0,Y 594.338,Z 530.536,A -85,B 0,C 180,E1 -1160.986,E2 -1160.986} C_VEL
LIN {X 0,Y 594.31,Z 537.613,A -85,B 0,C 180,E1 -1162.184,E2 -1162.184} C_VEL
LIN {X 0,Y 594.262,Z 544.491,A -85,B 0,C 180,E1 -1163.623,E2 -1163.623} C_VEL
LIN {X 0,Y 594.245,Z 549.325,A -85,B 0,C 180,E1 -1164.911,E2 -1164.911} C_VEL
LIN {X 0,Y 594.251,Z 552.289,A -85,B 0,C 180,E1 -1165.931,E2 -1165.931} C_VEL
LIN {X 0,Y 594.223,Z 555.186,A -85,B 0,C 180,E1 -1167.289,E2 -1167.289} C_VEL
LIN {X 0,Y 594.245,Z 556.913,A -85,B 0,C 180,E1 -1168.645,E2 -1168.645} C_VEL
LIN {X 0,Y 594.233,Z 557.5,A -85,B 0,C 180,E1 -1170,E2 -1170} C_VEL
LIN {X 0,Y 594.245,Z 556.912,A -85,B 0,C 180,E1 -1171.356,E2 -1171.356} C_VEL
LIN {X 0,Y 594.223,Z 555.185,A -85,B 0,C 180,E1 -1172.712,E2 -1172.712} C_VEL
LIN {X 0,Y 594.251,Z 552.287,A -85,B 0,C 180,E1 -1174.069,E2 -1174.069} C_VEL
LIN {X 0,Y 594.274,Z 548.161,A -85,B 0,C 180,E1 -1175.429,E2 -1175.429} C_VEL
LIN {X 0,Y 594.275,Z 542.702,A -85,B 0,C 180,E1 -1176.792,E2 -1176.792} C_VEL
LIN {X 0,Y 594.323,Z 535.749,A -85,B 0,C 180,E1 -1178.158,E2 -1178.158} C_VEL
LIN {X 0,Y 594.341,Z 527.089,A -85,B 0,C 180,E1 -1179.529,E2 -1179.529} C_VEL
LIN {X 0,Y 594.402,Z 517.874,A -85,B 0,C 180,E1 -1180.733,E2 -1180.733} C_VEL
LIN {X 0,Y 594.467,Z 508.506,A -85,B 0,C 180,E1 -1181.767,E2 -1181.767} C_VEL
LIN {X 0,Y 594.552,Z 497.385,A -85,B 0,C 180,E1 -1182.806,E2 -1182.806} C_VEL
LIN {X 0,Y 594.652,Z 484.642,A -85,B 0,C 180,E1 -1183.799,E2 -1183.799} C_VEL
LIN {X 0,Y 594.748,Z 471.778,A -85,B 0,C 180,E1 -1184.631,E2 -1184.631} C_VEL
LIN {X 0,Y 594.847,Z 458.603,A -85,B 0,C 180,E1 -1185.329,E2 -1185.329} C_VEL
LIN {X 0,Y 594.919,Z 444.176,A -85,B 0,C 180,E1 -1185.942,E2 -1185.942} C_VEL
LIN {X 0,Y 595.009,Z 429.243,A -85,B 0,C 180,E1 -1186.424,E2 -1186.424} C_VEL
LIN {X 0,Y 595.05,Z 413.815,A -85,B 0,C 180,E1 -1186.774,E2 -1186.774} C_VEL
LIN {X 0,Y 594.892,Z 404.357,A -85,B 0,C 180,E1 -1186.925,E2 -1186.925} C_VEL
LIN {X 0,Y 594.322,Z 401.716,A -85,B 0,C 180,E1 -1186.982,E2 -1186.982} C_VEL
LIN {X 0,Y 594.355,Z 392.838,A -85,B 0,C 180,E1 -1189.694,E2 -1189.694} C_VEL
LIN {X 0,Y 594.38,Z 384.666,A -85,B 0,C 180,E1 -1192.233,E2 -1192.233} C_VEL
LIN {X 0,Y 594.435,Z 375.325,A -85,B 0,C 180,E1 -1195.191,E2 -1195.191} C_VEL
LIN {X 0,Y 594.427,Z 367.149,A -85,B 0,C 180,E1 -1197.842,E2 -1197.842} C_VEL
LIN {X 0,Y 594.485,Z 359.603,A -85,B 0,C 180,E1 -1200.344,E2 -1200.344} C_VEL
LIN {X 0,Y 594.511,Z 351.849,A -85,B 0,C 180,E1 -1202.942,E2 -1202.942} C_VEL
LIN {X 0,Y 594.526,Z 344.683,A -85,B 0,C 180,E1 -1205.397,E2 -1205.397} C_VEL
LIN {X 0,Y 594.553,Z 337.525,A -85,B 0,C 180,E1 -1207.929,E2 -1207.929} C_VEL
LIN {X 0,Y 594.635,Z 329.827,A -85,B 0,C 180,E1 -1210.851,E2 -1210.851} C_VEL
LIN {X 0,Y 594.37,Z 327.076,A -85,B 0,C 180,E1 -1212.012,E2 -1212.012} C_VEL
LIN {X 0,Y 594.366,Z 327.072,A -85,B 0,C 180,E1 -1214.809,E2 -1214.809} C_VEL
LIN {X 0,Y 594.368,Z 327.073,A -85,B 0,C 180,E1 -1217.625,E2 -1217.625} C_VEL
LIN {X 0,Y 594.377,Z 327.075,A -85,B 0,C 180,E1 -1220.32,E2 -1220.32} C_VEL
LIN {X 0,Y 594.388,Z 327.071,A -85,B 0,C 180,E1 -1222.914,E2 -1222.914} C_VEL
LIN {X 0,Y 594.385,Z 327.071,A -85,B 0,C 180,E1 -1225.861,E2 -1225.861} C_VEL
LIN {X 0,Y 594.372,Z 327.071,A -85,B 0,C 180,E1 -1228.65,E2 -1228.65} C_VEL
LIN {X 0,Y 594.384,Z 327.073,A -85,B 0,C 180,E1 -1231.043,E2 -1231.043} C_VEL
LIN {X 0,Y 594.387,Z 327.069,A -85,B 0,C 180,E1 -1233.301,E2 -1233.301} C_VEL
LIN {X 0,Y 594.379,Z 327.07,A -85,B 0,C 180,E1 -1236.296,E2 -1236.296} C_VEL
LIN {X 0,Y 594.401,Z 327.067,A -85,B 0,C 180,E1 -1239.224,E2 -1239.224} C_VEL
LIN {X 0,Y 594.355,Z 327.074,A -85,B 0,C 180,E1 -1242.095,E2 -1242.095} C_VEL
LIN {X 0,Y 594.37,Z 327.073,A -85,B 0,C 180,E1 -1244.219,E2 -1244.219} C_VEL
LIN {X 0,Y 594.371,Z 327.071,A -85,B 0,C 180,E1 -1247.017,E2 -1247.017} C_VEL
LIN {X 0,Y 594.393,Z 327.069,A -85,B 0,C 180,E1 -1249.784,E2 -1249.784} C_VEL
LIN {X 0,Y 594.397,Z 327.07,A -85,B 0,C 180,E1 -1252.527,E2 -1252.527} C_VEL
LIN {X 0,Y 594.4,Z 327.074,A -85,B 0,C 180,E1 -1255.253,E2 -1255.253} C_VEL
LIN {X 0,Y 594.397,Z 327.07,A -85,B 0,C 180,E1 -1257.967,E2 -1257.967} C_VEL
LIN {X 0,Y 594.423,Z 327.065,A -85,B 0,C 180,E1 -1260.678,E2 -1260.678} C_VEL
LIN {X 0,Y 594.385,Z 327.07,A -85,B 0,C 180,E1 -1263.389,E2 -1263.389} C_VEL
LIN {X 0,Y 594.379,Z 327.073,A -85,B 0,C 180,E1 -1266.109,E2 -1266.109} C_VEL
LIN {X 0,Y 594.403,Z 327.072,A -85,B 0,C 180,E1 -1268.842,E2 -1268.842} C_VEL
LIN {X 0,Y 594.398,Z 327.068,A -85,B 0,C 180,E1 -1271.596,E2 -1271.596} C_VEL
LIN {X 0,Y 594.393,Z 327.068,A -85,B 0,C 180,E1 -1274.377,E2 -1274.377} C_VEL
LIN {X 0,Y 594.363,Z 327.074,A -85,B 0,C 180,E1 -1275.323,E2 -1275.323} C_VEL
LIN {X 0,Y 593.693,Z 327.156,A -85,B 0,C 180,E1 -1275.889,E2 -1275.889} C_VEL
LIN {X 0,Y 590.839,Z 327.515,A -85,B 0,C 180,E1 -1276.807,E2 -1276.807} C_VEL
LIN {X 0,Y 588.434,Z 327.817,A -85,B 0,C 180,E1 -1277.546,E2 -1277.546} C_VEL
LIN {X 0,Y 587.406,Z 327.944,A -85,B 0,C 180,E1 -1278.116,E2 -1278.116} C_VEL
LIN {X 0,Y 587.325,Z 327.951,A -85,B 0,C 180,E1 -1278.309,E2 -1278.309} C_VEL
LIN {X 0,Y 587.334,Z 327.95,A -85,B 0,C 180,E1 -1281.038,E2 -1281.038} C_VEL
LIN {X 0,Y 587.318,Z 327.95,A -85,B 0,C 180,E1 -1283.259,E2 -1283.259} C_VEL
LIN {X 0,Y 587.341,Z 327.95,A -85,B 0,C 180,E1 -1285.516,E2 -1285.516} C_VEL
LIN {X 0,Y 587.35,Z 327.945,A -85,B 0,C 180,E1 -1287.818,E2 -1287.818} C_VEL
LIN {X 0,Y 587.343,Z 327.95,A -85,B 0,C 180,E1 -1290.51,E2 -1290.51} C_VEL
LIN {X 0,Y 587.338,Z 327.952,A -85,B 0,C 180,E1 -1293.397,E2 -1293.397} C_VEL
LIN {X 0,Y 587.323,Z 327.95,A -85,B 0,C 180,E1 -1295.898,E2 -1295.898} C_VEL
LIN {X 0,Y 587.336,Z 327.948,A -85,B 0,C 180,E1 -1298.479,E2 -1298.479} C_VEL
LIN {X 0,Y 587.338,Z 327.951,A -85,B 0,C 180,E1 -1301.157,E2 -1301.157} C_VEL
LIN {X 0,Y 587.33,Z 327.953,A -85,B 0,C 180,E1 -1304.113,E2 -1304.113} C_VEL
LIN {X 0,Y 587.321,Z 327.955,A -85,B 0,C 180,E1 -1306.994,E2 -1306.994} C_VEL
LIN {X 0,Y 587.28,Z 327.961,A -85,B 0,C 180,E1 -1308.931,E2 -1308.931} C_VEL
LIN {X 0,Y 587.28,Z 330.598,A -85,B 0,C 180,E1 -1311.516,E2 -1311.516} C_VEL
LIN {X 0,Y 587.244,Z 333.581,A -85,B 0,C 180,E1 -1314.47,E2 -1314.47} C_VEL
LIN {X 0,Y 587.243,Z 336.073,A -85,B 0,C 180,E1 -1316.903,E2 -1316.903} C_VEL
LIN {X 0,Y 587.198,Z 339.153,A -85,B 0,C 180,E1 -1319.822,E2 -1319.822} C_VEL
LIN {X 0,Y 587.196,Z 342.029,A -85,B 0,C 180,E1 -1322.336,E2 -1322.336} C_VEL
LIN {X 0,Y 587.194,Z 345.822,A -85,B 0,C 180,E1 -1325.454,E2 -1325.454} C_VEL
LIN {X 0,Y 587.14,Z 349.268,A -85,B 0,C 180,E1 -1328.218,E2 -1328.218} C_VEL
LIN {X 0,Y 587.151,Z 352.819,A -85,B 0,C 180,E1 -1331.015,E2 -1331.015} C_VEL
LIN {X 0,Y 587.144,Z 355.249,A -85,B 0,C 180,E1 -1332.901,E2 -1332.901} C_VEL
LIN {X 0,Y 588.299,Z 360.903,A -85,B 0,C 180,E1 -1333.021,E2 -1333.021} C_VEL
LIN {X 0,Y 588.227,Z 375.905,A -85,B 0,C 180,E1 -1333.336,E2 -1333.336} C_VEL
LIN {X 0,Y 588.097,Z 390.483,A -85,B 0,C 180,E1 -1333.779,E2 -1333.779} C_VEL
LIN {X 0,Y 588.007,Z 403.79,A -85,B 0,C 180,E1 -1334.311,E2 -1334.311} C_VEL
LIN {X 0,Y 587.841,Z 417.871,A -85,B 0,C 180,E1 -1335.016,E2 -1335.016} C_VEL
LIN {X 0,Y 587.723,Z 431.182,A -85,B 0,C 180,E1 -1335.84,E2 -1335.84} C_VEL
LIN {X 0,Y 587.569,Z 443.683,A -85,B 0,C 180,E1 -1336.776,E2 -1336.776} C_VEL
LIN {X 0,Y 587.504,Z 454.513,A -85,B 0,C 180,E1 -1337.741,E2 -1337.741} C_VEL
LIN {X 0,Y 587.395,Z 464.993,A -85,B 0,C 180,E1 -1338.845,E2 -1338.845} C_VEL
LIN {X 0,Y 587.335,Z 474.296,A -85,B 0,C 180,E1 -1340.008,E2 -1340.008} C_VEL
LIN {X 0,Y 587.269,Z 482.454,A -85,B 0,C 180,E1 -1341.223,E2 -1341.223} C_VEL
LIN {X 0,Y 587.231,Z 489.187,A -85,B 0,C 180,E1 -1342.435,E2 -1342.435} C_VEL
LIN {X 0,Y 587.181,Z 495.421,A -85,B 0,C 180,E1 -1343.816,E2 -1343.816} C_VEL
LIN {X 0,Y 587.134,Z 500.245,A -85,B 0,C 180,E1 -1345.193,E2 -1345.193} C_VEL
LIN {X 0,Y 587.179,Z 503.792,A -85,B 0,C 180,E1 -1346.569,E2 -1346.569} C_VEL
LIN {X 0,Y 587.14,Z 506.14,A -85,B 0,C 180,E1 -1347.942,E2 -1347.942} C_VEL
LIN {X 0,Y 587.135,Z 507.337,A -85,B 0,C 180,E1 -1349.314,E2 -1349.314} C_VEL
LIN {X 0,Y 587.136,Z 507.36,A -85,B 0,C 180,E1 -1350.686,E2 -1350.686} C_VEL
LIN {X 0,Y 587.14,Z 506.245,A -85,B 0,C 180,E1 -1352.058,E2 -1352.058} C_VEL
LIN {X 0,Y 587.181,Z 503.982,A -85,B 0,C 180,E1 -1353.431,E2 -1353.431} C_VEL
LIN {X 0,Y 587.134,Z 500.523,A -85,B 0,C 180,E1 -1354.806,E2 -1354.806} C_VEL
LIN {X 0,Y 587.183,Z 495.794,A -85,B 0,C 180,E1 -1356.184,E2 -1356.184} C_VEL
LIN {X 0,Y 587.23,Z 489.662,A -85,B 0,C 180,E1 -1357.565,E2 -1357.565} C_VEL
LIN {X 0,Y 587.266,Z 481.944,A -85,B 0,C 180,E1 -1358.95,E2 -1358.95} C_VEL
LIN {X 0,Y 587.351,Z 473.702,A -85,B 0,C 180,E1 -1360.165,E2 -1360.165} C_VEL
LIN {X 0,Y 587.397,Z 463.799,A -85,B 0,C 180,E1 -1361.385,E2 -1361.385} C_VEL
LIN {X 0,Y 587.5,Z 453.651,A -85,B 0,C 180,E1 -1362.434,E2 -1362.434} C_VEL
LIN {X 0,Y 587.621,Z 441.579,A -85,B 0,C 180,E1 -1363.487,E2 -1363.487} C_VEL
LIN {X 0,Y 587.774,Z 427.926,A -85,B 0,C 180,E1 -1364.469,E2 -1364.469} C_VEL
LIN {X 0,Y 587.888,Z 414.744,A -85,B 0,C 180,E1 -1365.248,E2 -1365.248} C_VEL
LIN {X 0,Y 588.029,Z 399.815,A -85,B 0,C 180,E1 -1365.955,E2 -1365.955} C_VEL
LIN {X 0,Y 588.188,Z 385.318,A -85,B 0,C 180,E1 -1366.485,E2 -1366.485} C_VEL
LIN {X 0,Y 588.253,Z 369.675,A -85,B 0,C 180,E1 -1366.904,E2 -1366.904} C_VEL
LIN {X 0,Y 588.203,Z 359.916,A -85,B 0,C 180,E1 -1367.087,E2 -1367.087} C_VEL
LIN {X 0,Y 587.152,Z 355.23,A -85,B 0,C 180,E1 -1367.203,E2 -1367.203} C_VEL
LIN {X 0,Y 587.131,Z 352.171,A -85,B 0,C 180,E1 -1369.582,E2 -1369.582} C_VEL
LIN {X 0,Y 587.138,Z 349.382,A -85,B 0,C 180,E1 -1371.781,E2 -1371.781} C_VEL
LIN {X 0,Y 587.176,Z 345.663,A -85,B 0,C 180,E1 -1374.766,E2 -1374.766} C_VEL
LIN {X 0,Y 587.16,Z 342.873,A -85,B 0,C 180,E1 -1377.054,E2 -1377.054} C_VEL
LIN {X 0,Y 587.163,Z 340.1,A -85,B 0,C 180,E1 -1379.389,E2 -1379.389} C_VEL
LIN {X 0,Y 587.219,Z 337.522,A -85,B 0,C 180,E1 -1381.816,E2 -1381.816} C_VEL
LIN {X 0,Y 587.246,Z 334.909,A -85,B 0,C 180,E1 -1384.333,E2 -1384.333} C_VEL
LIN {X 0,Y 587.261,Z 332.448,A -85,B 0,C 180,E1 -1386.753,E2 -1386.753} C_VEL
LIN {X 0,Y 587.246,Z 329.775,A -85,B 0,C 180,E1 -1389.367,E2 -1389.367} C_VEL
LIN {X 0,Y 587.284,Z 327.96,A -85,B 0,C 180,E1 -1391.161,E2 -1391.161} C_VEL
LIN {X 0,Y 587.326,Z 327.953,A -85,B 0,C 180,E1 -1393.119,E2 -1393.119} C_VEL
LIN {X 0,Y 587.323,Z 327.955,A -85,B 0,C 180,E1 -1396.049,E2 -1396.049} C_VEL
LIN {X 0,Y 587.335,Z 327.951,A -85,B 0,C 180,E1 -1398.925,E2 -1398.925} C_VEL
LIN {X 0,Y 587.333,Z 327.948,A -85,B 0,C 180,E1 -1401.521,E2 -1401.521} C_VEL
LIN {X 0,Y 587.352,Z 327.945,A -85,B 0,C 180,E1 -1404.454,E2 -1404.454} C_VEL
LIN {X 0,Y 587.336,Z 327.951,A -85,B 0,C 180,E1 -1406.888,E2 -1406.888} C_VEL
LIN {X 0,Y 587.351,Z 327.948,A -85,B 0,C 180,E1 -1409.487,E2 -1409.487} C_VEL
LIN {X 0,Y 587.351,Z 327.945,A -85,B 0,C 180,E1 -1412.307,E2 -1412.307} C_VEL
LIN {X 0,Y 587.34,Z 327.951,A -85,B 0,C 180,E1 -1414.484,E2 -1414.484} C_VEL
LIN {X 0,Y 587.318,Z 327.952,A -85,B 0,C 180,E1 -1417.131,E2 -1417.131} C_VEL
LIN {X 0,Y 587.329,Z 327.946,A -85,B 0,C 180,E1 -1419.695,E2 -1419.695} C_VEL
LIN {X 0,Y 587.359,Z 327.945,A -85,B 0,C 180,E1 -1422.594,E2 -1422.594} C_VEL
LIN {X 0,Y 587.364,Z 327.943,A -85,B 0,C 180,E1 -1425.739,E2 -1425.739} C_VEL
LIN {X 0,Y 587.346,Z 327.945,A -85,B 0,C 180,E1 -1428.866,E2 -1428.866} C_VEL
LIN {X 0,Y 587.369,Z 327.943,A -85,B 0,C 180,E1 -1431.745,E2 -1431.745} C_VEL
LIN {X 0,Y 587.361,Z 327.946,A -85,B 0,C 180,E1 -1434.507,E2 -1434.507} C_VEL
LIN {X 0,Y 587.381,Z 327.947,A -85,B 0,C 180,E1 -1437.257,E2 -1437.257} C_VEL
LIN {X 0,Y 587.38,Z 327.945,A -85,B 0,C 180,E1 -1440,E2 -1440} C_VEL
LIN {X 0,Y 587.378,Z 327.943,A -85,B 0,C 180,E1 -1442.743,E2 -1442.743} C_VEL
LIN {X 0,Y 587.359,Z 327.945,A -85,B 0,C 180,E1 -1445.493,E2 -1445.493} C_VEL
LIN {X 0,Y 587.367,Z 327.945,A -85,B 0,C 180,E1 -1448.255,E2 -1448.255} C_VEL
LIN {X 0,Y 587.362,Z 327.947,A -85,B 0,C 180,E1 -1451.141,E2 -1451.141} C_VEL
LIN {X 0,Y 587.364,Z 327.946,A -85,B 0,C 180,E1 -1454.261,E2 -1454.261} C_VEL
LIN {X 0,Y 587.351,Z 327.947,A -85,B 0,C 180,E1 -1457.406,E2 -1457.406} C_VEL
LIN {X 0,Y 587.327,Z 327.951,A -85,B 0,C 180,E1 -1460.305,E2 -1460.305} C_VEL
LIN {X 0,Y 587.321,Z 327.953,A -85,B 0,C 180,E1 -1463.259,E2 -1463.259} C_VEL
LIN {X 0,Y 587.331,Z 327.948,A -85,B 0,C 180,E1 -1465.517,E2 -1465.517} C_VEL
LIN {X 0,Y 587.347,Z 327.95,A -85,B 0,C 180,E1 -1467.818,E2 -1467.818} C_VEL
LIN {X 0,Y 587.35,Z 327.95,A -85,B 0,C 180,E1 -1470.513,E2 -1470.513} C_VEL
LIN {X 0,Y 587.333,Z 327.95,A -85,B 0,C 180,E1 -1473.397,E2 -1473.397} C_VEL
LIN {X 0,Y 587.356,Z 327.945,A -85,B 0,C 180,E1 -1475.895,E2 -1475.895} C_VEL
LIN {X 0,Y 587.334,Z 327.951,A -85,B 0,C 180,E1 -1478.479,E2 -1478.479} C_VEL
LIN {X 0,Y 587.337,Z 327.952,A -85,B 0,C 180,E1 -1481.157,E2 -1481.157} C_VEL
LIN {X 0,Y 587.325,Z 327.952,A -85,B 0,C 180,E1 -1484.114,E2 -1484.114} C_VEL
LIN {X 0,Y 587.322,Z 327.953,A -85,B 0,C 180,E1 -1486.995,E2 -1486.995} C_VEL
LIN {X 0,Y 587.366,Z 328.08,A -85,B 0,C 180,E1 -1487.825,E2 -1487.825} C_VEL
LIN {X 0,Y 587.688,Z 331.69,A -85,B 0,C 180,E1 -1489.336,E2 -1489.336} C_VEL
LIN {X 0,Y 587.577,Z 339.8,A -85,B 0,C 180,E1 -1492.41,E2 -1492.41} C_VEL
LIN {X 0,Y 587.533,Z 346.927,A -85,B 0,C 180,E1 -1494.959,E2 -1494.959} C_VEL
LIN {X 0,Y 587.537,Z 355.248,A -85,B 0,C 180,E1 -1497.823,E2 -1497.823} C_VEL
LIN {X 0,Y 587.483,Z 363.652,A -85,B 0,C 180,E1 -1500.628,E2 -1500.628} C_VEL
LIN {X 0,Y 587.432,Z 372.992,A -85,B 0,C 180,E1 -1503.726,E2 -1503.726} C_VEL
LIN {X 0,Y 587.379,Z 382.333,A -85,B 0,C 180,E1 -1506.744,E2 -1506.744} C_VEL
LIN {X 0,Y 587.314,Z 391.673,A -85,B 0,C 180,E1 -1509.695,E2 -1509.695} C_VEL
LIN {X 0,Y 587.286,Z 399.845,A -85,B 0,C 180,E1 -1512.233,E2 -1512.233} C_VEL
LIN {X 0,Y 587.274,Z 401.798,A -85,B 0,C 180,E1 -1512.816,E2 -1512.816} C_VEL
LIN {X 0,Y 588.304,Z 406.689,A -85,B 0,C 180,E1 -1512.914,E2 -1512.914} C_VEL
LIN {X 0,Y 588.257,Z 421.917,A -85,B 0,C 180,E1 -1513.195,E2 -1513.195} C_VEL
LIN {X 0,Y 588.155,Z 436.621,A -85,B 0,C 180,E1 -1513.603,E2 -1513.603} C_VEL
LIN {X 0,Y 588.005,Z 450.846,A -85,B 0,C 180,E1 -1514.133,E2 -1514.133} C_VEL
LIN {X 0,Y 587.874,Z 465.53,A -85,B 0,C 180,E1 -1514.84,E2 -1514.84} C_VEL
LIN {X 0,Y 587.756,Z 478.17,A -85,B 0,C 180,E1 -1515.591,E2 -1515.591} C_VEL
LIN {X 0,Y 587.629,Z 491.019,A -85,B 0,C 180,E1 -1516.514,E2 -1516.514} C_VEL
LIN {X 0,Y 587.521,Z 503.194,A -85,B 0,C 180,E1 -1517.566,E2 -1517.566} C_VEL
LIN {X 0,Y 587.424,Z 513.708,A -85,B 0,C 180,E1 -1518.65,E2 -1518.65} C_VEL
LIN {X 0,Y 587.351,Z 523.372,A -85,B 0,C 180,E1 -1519.835,E2 -1519.835} C_VEL
LIN {X 0,Y 587.266,Z 531.655,A -85,B 0,C 180,E1 -1521.05,E2 -1521.05} C_VEL
LIN {X 0,Y 587.229,Z 539.427,A -85,B 0,C 180,E1 -1522.435,E2 -1522.435} C_VEL
LIN {X 0,Y 587.18,Z 545.608,A -85,B 0,C 180,E1 -1523.816,E2 -1523.816} C_VEL
LIN {X 0,Y 587.136,Z 550.385,A -85,B 0,C 180,E1 -1525.194,E2 -1525.194} C_VEL
LIN {X 0,Y 587.179,Z 553.888,A -85,B 0,C 180,E1 -1526.569,E2 -1526.569} C_VEL
LIN {X 0,Y 587.14,Z 556.193,A -85,B 0,C 180,E1 -1527.942,E2 -1527.942} C_VEL
LIN {X 0,Y 587.137,Z 557.35,A -85,B 0,C 180,E1 -1529.314,E2 -1529.314} C_VEL
LIN {X 0,Y 587.137,Z 557.35,A -85,B 0,C 180,E1 -1530.686,E2 -1530.686} C_VEL
LIN {X 0,Y 587.14,Z 556.192,A -85,B 0,C 180,E1 -1532.058,E2 -1532.058} C_VEL
LIN {X 0,Y 587.179,Z 553.886,A -85,B 0,C 180,E1 -1533.431,E2 -1533.431} C_VEL
LIN {X 0,Y 587.136,Z 550.383,A -85,B 0,C 180,E1 -1534.807,E2 -1534.807} C_VEL
LIN {X 0,Y 587.18,Z 545.607,A -85,B 0,C 180,E1 -1536.184,E2 -1536.184} C_VEL
LIN {X 0,Y 587.23,Z 539.423,A -85,B 0,C 180,E1 -1537.565,E2 -1537.565} C_VEL
LIN {X 0,Y 587.266,Z 531.649,A -85,B 0,C 180,E1 -1538.95,E2 -1538.95} C_VEL
LIN {X 0,Y 587.351,Z 523.368,A -85,B 0,C 180,E1 -1540.166,E2 -1540.166} C_VEL
LIN {X 0,Y 587.4,Z 513.392,A -85,B 0,C 180,E1 -1541.386,E2 -1541.386} C_VEL
LIN {X 0,Y 587.522,Z 503.188,A -85,B 0,C 180,E1 -1542.434,E2 -1542.434} C_VEL
LIN {X 0,Y 587.629,Z 491.014,A -85,B 0,C 180,E1 -1543.487,E2 -1543.487} C_VEL
LIN {X 0,Y 587.775,Z 478.05,A -85,B 0,C 180,E1 -1544.416,E2 -1544.416} C_VEL
LIN {X 0,Y 587.875,Z 465.517,A -85,B 0,C 180,E1 -1545.16,E2 -1545.16} C_VEL
LIN {X 0,Y 588.005,Z 450.832,A -85,B 0,C 180,E1 -1545.867,E2 -1545.867} C_VEL
LIN {X 0,Y 588.156,Z 436.608,A -85,B 0,C 180,E1 -1546.398,E2 -1546.398} C_VEL
LIN {X 0,Y 588.251,Z 421.387,A -85,B 0,C 180,E1 -1546.818,E2 -1546.818} C_VEL
LIN {X 0,Y 588.237,Z 406.069,A -85,B 0,C 180,E1 -1547.098,E2 -1547.098} C_VEL
LIN {X 0,Y 587.249,Z 401.675,A -85,B 0,C 180,E1 -1547.205,E2 -1547.205} C_VEL
LIN {X 0,Y 587.32,Z 392.838,A -85,B 0,C 180,E1 -1549.94,E2 -1549.94} C_VEL
LIN {X 0,Y 587.334,Z 384.666,A -85,B 0,C 180,E1 -1552.514,E2 -1552.514} C_VEL
LIN {X 0,Y 587.418,Z 375.325,A -85,B 0,C 180,E1 -1555.513,E2 -1555.513} C_VEL
LIN {X 0,Y 587.474,Z 365.985,A -85,B 0,C 180,E1 -1558.589,E2 -1558.589} C_VEL
LIN {X 0,Y 587.473,Z 357.702,A -85,B 0,C 180,E1 -1561.359,E2 -1561.359} C_VEL
LIN {X 0,Y 587.526,Z 350.485,A -85,B 0,C 180,E1 -1563.796,E2 -1563.796} C_VEL
LIN {X 0,Y 587.567,Z 342.132,A -85,B 0,C 180,E1 -1566.736,E2 -1566.736} C_VEL
LIN {X 0,Y 587.593,Z 335.088,A -85,B 0,C 180,E1 -1569.34,E2 -1569.34} C_VEL
LIN {X 0,Y 587.63,Z 330.545,A -85,B 0,C 180,E1 -1571.132,E2 -1571.132} C_VEL
LIN {X 0,Y 587.327,Z 327.954,A -85,B 0,C 180,E1 -1572.306,E2 -1572.306} C_VEL
LIN {X 0,Y 587.319,Z 327.951,A -85,B 0,C 180,E1 -1575.089,E2 -1575.089} C_VEL
LIN {X 0,Y 587.326,Z 327.949,A -85,B 0,C 180,E1 -1577.925,E2 -1577.925} C_VEL
LIN {X 0,Y 587.338,Z 327.949,A -85,B 0,C 180,E1 -1580.64,E2 -1580.64} C_VEL
LIN {X 0,Y 587.357,Z 327.951,A -85,B 0,C 180,E1 -1583.292,E2 -1583.292} C_VEL
LIN {X 0,Y 587.367,Z 327.945,A -85,B 0,C 180,E1 -1585.78,E2 -1585.78} C_VEL
LIN {X 0,Y 587.342,Z 327.948,A -85,B 0,C 180,E1 -1588.231,E2 -1588.231} C_VEL
LIN {X 0,Y 587.351,Z 327.952,A -85,B 0,C 180,E1 -1590.867,E2 -1590.867} C_VEL
LIN {X 0,Y 587.339,Z 327.951,A -85,B 0,C 180,E1 -1593.722,E2 -1593.722} C_VEL
LIN {X 0,Y 587.332,Z 327.948,A -85,B 0,C 180,E1 -1595.993,E2 -1595.993} C_VEL
LIN {X 0,Y 587.325,Z 327.952,A -85,B 0,C 180,E1 -1598.226,E2 -1598.226} C_VEL
LIN {X 0,Y 587.351,Z 327.947,A -85,B 0,C 180,E1 -1601.151,E2 -1601.151} C_VEL
LIN {X 0,Y 587.328,Z 327.949,A -85,B 0,C 180,E1 -1604.025,E2 -1604.025} C_VEL
LIN {X 0,Y 587.365,Z 327.95,A -85,B 0,C 180,E1 -1606.154,E2 -1606.154} C_VEL
LIN {X 0,Y 587.349,Z 327.95,A -85,B 0,C 180,E1 -1608.963,E2 -1608.963} C_VEL
LIN {X 0,Y 587.368,Z 327.944,A -85,B 0,C 180,E1 -1611.745,E2 -1611.745} C_VEL
LIN {X 0,Y 587.358,Z 327.945,A -85,B 0,C 180,E1 -1614.507,E2 -1614.507} C_VEL
LIN {X 0,Y 587.38,Z 327.943,A -85,B 0,C 180,E1 -1617.257,E2 -1617.257} C_VEL
LIN {X 0,Y 587.384,Z 327.945,A -85,B 0,C 180,E1 -1620,E2 -1620} C_VEL
LIN {X 0,Y 587.382,Z 327.946,A -85,B 0,C 180,E1 -1622.743,E2 -1622.743} C_VEL
LIN {X 0,Y 587.363,Z 327.945,A -85,B 0,C 180,E1 -1625.493,E2 -1625.493} C_VEL
LIN {X 0,Y 587.371,Z 327.943,A -85,B 0,C 180,E1 -1628.255,E2 -1628.255} C_VEL
LIN {X 0,Y 587.352,Z 327.944,A -85,B 0,C 180,E1 -1631.134,E2 -1631.134} C_VEL
LIN {X 0,Y 587.368,Z 327.942,A -85,B 0,C 180,E1 -1634.26,E2 -1634.26} C_VEL
LIN {X 0,Y 587.361,Z 327.944,A -85,B 0,C 180,E1 -1637.406,E2 -1637.406} C_VEL
LIN {X 0,Y 587.325,Z 327.951,A -85,B 0,C 180,E1 -1638.309,E2 -1638.309} C_VEL
LIN {X 0,Y 586.671,Z 328.029,A -85,B 0,C 180,E1 -1638.881,E2 -1638.881} C_VEL
LIN {X 0,Y 583.842,Z 328.386,A -85,B 0,C 180,E1 -1639.81,E2 -1639.81} C_VEL
LIN {X 0,Y 581.434,Z 328.689,A -85,B 0,C 180,E1 -1640.557,E2 -1640.557} C_VEL
LIN {X 0,Y 580.382,Z 328.818,A -85,B 0,C 180,E1 -1641.133,E2 -1641.133} C_VEL
LIN {X 0,Y 580.287,Z 328.828,A -85,B 0,C 180,E1 -1641.328,E2 -1641.328} C_VEL
LIN {X 0,Y 580.302,Z 328.828,A -85,B 0,C 180,E1 -1644.316,E2 -1644.316} C_VEL
LIN {X 0,Y 580.282,Z 328.825,A -85,B 0,C 180,E1 -1646.623,E2 -1646.623} C_VEL
LIN {X 0,Y 580.305,Z 328.823,A -85,B 0,C 180,E1 -1649.31,E2 -1649.31} C_VEL
LIN {X 0,Y 580.301,Z 328.824,A -85,B 0,C 180,E1 -1652.2,E2 -1652.2} C_VEL
LIN {X 0,Y 580.295,Z 328.827,A -85,B 0,C 180,E1 -1654.696,E2 -1654.696} C_VEL
LIN {X 0,Y 580.303,Z 328.824,A -85,B 0,C 180,E1 -1657.268,E2 -1657.268} C_VEL
LIN {X 0,Y 580.299,Z 328.824,A -85,B 0,C 180,E1 -1660.271,E2 -1660.271} C_VEL
LIN {X 0,Y 580.28,Z 328.83,A -85,B 0,C 180,E1 -1662.706,E2 -1662.706} C_VEL
LIN {X 0,Y 580.273,Z 328.833,A -85,B 0,C 180,E1 -1665.609,E2 -1665.609} C_VEL
LIN {X 0,Y 580.272,Z 328.83,A -85,B 0,C 180,E1 -1668.23,E2 -1668.23} C_VEL
LIN {X 0,Y 580.2,Z 328.896,A -85,B 0,C 180,E1 -1669.148,E2 -1669.148} C_VEL
LIN {X 0,Y 580.209,Z 331.75,A -85,B 0,C 180,E1 -1671.938,E2 -1671.938} C_VEL
LIN {X 0,Y 580.2,Z 334.245,A -85,B 0,C 180,E1 -1674.449,E2 -1674.449} C_VEL
LIN {X 0,Y 580.189,Z 336.789,A -85,B 0,C 180,E1 -1676.968,E2 -1676.968} C_VEL
LIN {X 0,Y 580.138,Z 339.344,A -85,B 0,C 180,E1 -1679.416,E2 -1679.416} C_VEL
LIN {X 0,Y 580.102,Z 342.278,A -85,B 0,C 180,E1 -1682.178,E2 -1682.178} C_VEL
LIN {X 0,Y 580.084,Z 345.552,A -85,B 0,C 180,E1 -1684.91,E2 -1684.91} C_VEL
LIN {X 0,Y 580.074,Z 348.339,A -85,B 0,C 180,E1 -1687.188,E2 -1687.188} C_VEL
LIN {X 0,Y 580.085,Z 351.127,A -85,B 0,C 180,E1 -1689.43,E2 -1689.43} C_VEL
LIN {X 0,Y 580.041,Z 354.843,A -85,B 0,C 180,E1 -1692.367,E2 -1692.367} C_VEL
LIN {X 0,Y 580.07,Z 355.369,A -85,B 0,C 180,E1 -1692.688,E2 -1692.688} C_VEL
LIN {X 0,Y 581.526,Z 362.554,A -85,B 0,C 180,E1 -1692.844,E2 -1692.844} C_VEL
LIN {X 0,Y 581.417,Z 377.666,A -85,B 0,C 180,E1 -1693.179,E2 -1693.179} C_VEL
LIN {X 0,Y 581.244,Z 393.044,A -85,B 0,C 180,E1 -1693.673,E2 -1693.673} C_VEL
LIN {X 0,Y 581.096,Z 407.711,A -85,B 0,C 180,E1 -1694.299,E2 -1694.299} C_VEL
LIN {X 0,Y 580.927,Z 421.014,A -85,B 0,C 180,E1 -1695.013,E2 -1695.013} C_VEL
LIN {X 0,Y 580.792,Z 434.365,A -85,B 0,C 180,E1 -1695.89,E2 -1695.89} C_VEL
LIN {X 0,Y 580.591,Z 446.869,A -85,B 0,C 180,E1 -1696.881,E2 -1696.881} C_VEL
LIN {X 0,Y 580.461,Z 458.07,A -85,B 0,C 180,E1 -1697.944,E2 -1697.944} C_VEL
LIN {X 0,Y 580.337,Z 469.11,A -85,B 0,C 180,E1 -1699.201,E2 -1699.201} C_VEL
LIN {X 0,Y 580.239,Z 477.996,A -85,B 0,C 180,E1 -1700.413,E2 -1700.413} C_VEL
LIN {X 0,Y 580.195,Z 485.489,A -85,B 0,C 180,E1 -1701.642,E2 -1701.642} C_VEL
LIN {X 0,Y 580.139,Z 492.493,A -85,B 0,C 180,E1 -1703.042,E2 -1703.042} C_VEL
LIN {X 0,Y 580.127,Z 498.002,A -85,B 0,C 180,E1 -1704.438,E2 -1704.438} C_VEL
LIN {X 0,Y 580.087,Z 502.173,A -85,B 0,C 180,E1 -1705.831,E2 -1705.831} C_VEL
LIN {X 0,Y 580.038,Z 505.114,A -85,B 0,C 180,E1 -1707.222,E2 -1707.222} C_VEL
LIN {X 0,Y 580.043,Z 506.88,A -85,B 0,C 180,E1 -1708.611,E2 -1708.611} C_VEL
LIN {X 0,Y 580.035,Z 507.496,A -85,B 0,C 180,E1 -1710,E2 -1710} C_VEL
LIN {X 0,Y 580.045,Z 506.943,A -85,B 0,C 180,E1 -1711.388,E2 -1711.388} C_VEL
LIN {X 0,Y 580.04,Z 505.259,A -85,B 0,C 180,E1 -1712.778,E2 -1712.778} C_VEL
LIN {X 0,Y 580.087,Z 502.405,A -85,B 0,C 180,E1 -1714.168,E2 -1714.168} C_VEL
LIN {X 0,Y 580.123,Z 498.322,A -85,B 0,C 180,E1 -1715.561,E2 -1715.561} C_VEL
LIN {X 0,Y 580.138,Z 492.911,A -85,B 0,C 180,E1 -1716.958,E2 -1716.958} C_VEL
LIN {X 0,Y 580.19,Z 486.011,A -85,B 0,C 180,E1 -1718.358,E2 -1718.358} C_VEL
LIN {X 0,Y 580.235,Z 477.407,A -85,B 0,C 180,E1 -1719.763,E2 -1719.763} C_VEL
LIN {X 0,Y 580.308,Z 467.834,A -85,B 0,C 180,E1 -1721.046,E2 -1721.046} C_VEL
LIN {X 0,Y 580.472,Z 457.202,A -85,B 0,C 180,E1 -1722.232,E2 -1722.232} C_VEL
LIN {X 0,Y 580.606,Z 445.827,A -85,B 0,C 180,E1 -1723.296,E2 -1723.296} C_VEL
LIN {X 0,Y 580.77,Z 433.081,A -85,B 0,C 180,E1 -1724.29,E2 -1724.29} C_VEL
LIN {X 0,Y 580.952,Z 419.465,A -85,B 0,C 180,E1 -1725.165,E2 -1725.165} C_VEL
LIN {X 0,Y 581.128,Z 405.789,A -85,B 0,C 180,E1 -1725.879,E2 -1725.879} C_VEL
LIN {X 0,Y 581.271,Z 391.8,A -85,B 0,C 180,E1 -1726.462,E2 -1726.462} C_VEL
LIN {X 0,Y 581.44,Z 376.734,A -85,B 0,C 180,E1 -1726.934,E2 -1726.934} C_VEL
LIN {X 0,Y 581.428,Z 361.29,A -85,B 0,C 180,E1 -1727.271,E2 -1727.271} C_VEL
LIN {X 0,Y 580.048,Z 355.231,A -85,B 0,C 180,E1 -1727.419,E2 -1727.419} C_VEL
LIN {X 0,Y 580.061,Z 352.17,A -85,B 0,C 180,E1 -1729.831,E2 -1729.831} C_VEL
LIN {X 0,Y 580.041,Z 349.381,A -85,B 0,C 180,E1 -1732.062,E2 -1732.062} C_VEL
LIN {X 0,Y 580.093,Z 346.158,A -85,B 0,C 180,E1 -1734.681,E2 -1734.681} C_VEL
LIN {X 0,Y 580.085,Z 342.872,A -85,B 0,C 180,E1 -1737.412,E2 -1737.412} C_VEL
LIN {X 0,Y 580.104,Z 340.295,A -85,B 0,C 180,E1 -1739.783,E2 -1739.783} C_VEL
LIN {X 0,Y 580.136,Z 337.759,A -85,B 0,C 180,E1 -1742.21,E2 -1742.21} C_VEL
LIN {X 0,Y 580.163,Z 335.184,A -85,B 0,C 180,E1 -1744.704,E2 -1744.704} C_VEL
LIN {X 0,Y 580.197,Z 332.637,A -85,B 0,C 180,E1 -1747.276,E2 -1747.276} C_VEL
LIN {X 0,Y 580.188,Z 329.912,A -85,B 0,C 180,E1 -1749.941,E2 -1749.941} C_VEL
LIN {X 0,Y 580.202,Z 328.987,A -85,B 0,C 180,E1 -1750.851,E2 -1750.851} C_VEL
LIN {X 0,Y 580.286,Z 328.827,A -85,B 0,C 180,E1 -1753.391,E2 -1753.391} C_VEL
LIN {X 0,Y 580.279,Z 328.829,A -85,B 0,C 180,E1 -1756.342,E2 -1756.342} C_VEL
LIN {X 0,Y 580.298,Z 328.83,A -85,B 0,C 180,E1 -1759.156,E2 -1759.156} C_VEL
LIN {X 0,Y 580.29,Z 328.828,A -85,B 0,C 180,E1 -1761.927,E2 -1761.927} C_VEL
LIN {X 0,Y 580.307,Z 328.823,A -85,B 0,C 180,E1 -1764.456,E2 -1764.456} C_VEL
LIN {X 0,Y 580.288,Z 328.827,A -85,B 0,C 180,E1 -1766.975,E2 -1766.975} C_VEL
LIN {X 0,Y 580.31,Z 328.824,A -85,B 0,C 180,E1 -1769.426,E2 -1769.426} C_VEL
LIN {X 0,Y 580.319,Z 328.82,A -85,B 0,C 180,E1 -1772.137,E2 -1772.137} C_VEL
LIN {X 0,Y 580.309,Z 328.823,A -85,B 0,C 180,E1 -1774.92,E2 -1774.92} C_VEL
LIN {X 0,Y 580.272,Z 328.827,A -85,B 0,C 180,E1 -1777.947,E2 -1777.947} C_VEL
LIN {X 0,Y 580.318,Z 328.822,A -85,B 0,C 180,E1 -1780.914,E2 -1780.914} C_VEL
LIN {X 0,Y 580.281,Z 328.828,A -85,B 0,C 180,E1 -1783.826,E2 -1783.826} C_VEL
LIN {X 0,Y 580.326,Z 328.82,A -85,B 0,C 180,E1 -1785.983,E2 -1785.983} C_VEL
LIN {X 0,Y 580.303,Z 328.823,A -85,B 0,C 180,E1 -1788.827,E2 -1788.827} C_VEL
LIN {X 0,Y 580.333,Z 328.82,A -85,B 0,C 180,E1 -1791.644,E2 -1791.644} C_VEL
LIN {X 0,Y 580.328,Z 328.823,A -85,B 0,C 180,E1 -1794.44,E2 -1794.44} C_VEL
LIN {X 0,Y 580.346,Z 328.824,A -85,B 0,C 180,E1 -1797.223,E2 -1797.223} C_VEL
LIN {X 0,Y 580.35,Z 328.821,A -85,B 0,C 180,E1 -1800,E2 -1800} C_VEL
LIN {X 0,Y 580.343,Z 328.819,A -85,B 0,C 180,E1 -1802.776,E2 -1802.776} C_VEL
LIN {X 0,Y 580.324,Z 328.821,A -85,B 0,C 180,E1 -1805.56,E2 -1805.56} C_VEL
LIN {X 0,Y 580.329,Z 328.821,A -85,B 0,C 180,E1 -1808.356,E2 -1808.356} C_VEL
LIN {X 0,Y 580.333,Z 328.822,A -85,B 0,C 180,E1 -1811.208,E2 -1811.208} C_VEL
LIN {X 0,Y 580.314,Z 328.823,A -85,B 0,C 180,E1 -1814.339,E2 -1814.339} C_VEL
LIN {X 0,Y 580.311,Z 328.828,A -85,B 0,C 180,E1 -1816.914,E2 -1816.914} C_VEL
LIN {X 0,Y 580.304,Z 328.827,A -85,B 0,C 180,E1 -1819.822,E2 -1819.822} C_VEL
LIN {X 0,Y 580.293,Z 328.827,A -85,B 0,C 180,E1 -1822.802,E2 -1822.802} C_VEL
LIN {X 0,Y 580.305,Z 328.824,A -85,B 0,C 180,E1 -1825.08,E2 -1825.08} C_VEL
LIN {X 0,Y 580.299,Z 328.825,A -85,B 0,C 180,E1 -1828.185,E2 -1828.185} C_VEL
LIN {X 0,Y 580.299,Z 328.83,A -85,B 0,C 180,E1 -1830.697,E2 -1830.697} C_VEL
LIN {X 0,Y 580.301,Z 328.825,A -85,B 0,C 180,E1 -1833.317,E2 -1833.317} C_VEL
LIN {X 0,Y 580.325,Z 328.822,A -85,B 0,C 180,E1 -1835.768,E2 -1835.768} C_VEL
LIN {X 0,Y 580.289,Z 328.83,A -85,B 0,C 180,E1 -1838.146,E2 -1838.146} C_VEL
LIN {X 0,Y 580.3,Z 328.825,A -85,B 0,C 180,E1 -1840.843,E2 -1840.843} C_VEL
LIN {X 0,Y 580.277,Z 328.828,A -85,B 0,C 180,E1 -1843.658,E2 -1843.658} C_VEL
LIN {X 0,Y 580.285,Z 328.829,A -85,B 0,C 180,E1 -1846.608,E2 -1846.608} C_VEL
LIN {X 0,Y 580.312,Z 328.986,A -85,B 0,C 180,E1 -1847.59,E2 -1847.59} C_VEL
LIN {X 0,Y 580.732,Z 332.733,A -85,B 0,C 180,E1 -1849.194,E2 -1849.194} C_VEL
LIN {X 0,Y 580.595,Z 340.84,A -85,B 0,C 180,E1 -1852.323,E2 -1852.323} C_VEL
LIN {X 0,Y 580.546,Z 347.96,A -85,B 0,C 180,E1 -1854.899,E2 -1854.899} C_VEL
LIN {X 0,Y 580.513,Z 356.695,A -85,B 0,C 180,E1 -1857.936,E2 -1857.936} C_VEL
LIN {X 0,Y 580.474,Z 364.847,A -85,B 0,C 180,E1 -1860.66,E2 -1860.66} C_VEL
LIN {X 0,Y 580.4,Z 373.78,A -85,B 0,C 180,E1 -1863.644,E2 -1863.644} C_VEL
LIN {X 0,Y 580.315,Z 382.333,A -85,B 0,C 180,E1 -1866.444,E2 -1866.444} C_VEL
LIN {X 0,Y 580.265,Z 391.673,A -85,B 0,C 180,E1 -1869.437,E2 -1869.437} C_VEL
LIN {X 0,Y 580.207,Z 401.013,A -85,B 0,C 180,E1 -1872.373,E2 -1872.373} C_VEL
LIN {X 0,Y 580.19,Z 401.712,A -85,B 0,C 180,E1 -1872.591,E2 -1872.591} C_VEL
LIN {X 0,Y 581.537,Z 408.407,A -85,B 0,C 180,E1 -1872.734,E2 -1872.734} C_VEL
LIN {X 0,Y 581.414,Z 424.332,A -85,B 0,C 180,E1 -1873.051,E2 -1873.051} C_VEL
LIN {X 0,Y 581.311,Z 439.216,A -85,B 0,C 180,E1 -1873.495,E2 -1873.495} C_VEL
LIN {X 0,Y 581.13,Z 452.831,A -85,B 0,C 180,E1 -1874.03,E2 -1874.03} C_VEL
LIN {X 0,Y 580.984,Z 467.109,A -85,B 0,C 180,E1 -1874.746,E2 -1874.746} C_VEL
LIN {X 0,Y 580.799,Z 480.574,A -85,B 0,C 180,E1 -1875.58,E2 -1875.58} C_VEL
LIN {X 0,Y 580.629,Z 493.169,A -85,B 0,C 180,E1 -1876.526,E2 -1876.526} C_VEL
LIN {X 0,Y 580.515,Z 504.975,A -85,B 0,C 180,E1 -1877.591,E2 -1877.591} C_VEL
LIN {X 0,Y 580.335,Z 516.092,A -85,B 0,C 180,E1 -1878.792,E2 -1878.792} C_VEL
LIN {X 0,Y 580.268,Z 525.859,A -85,B 0,C 180,E1 -1880.062,E2 -1880.062} C_VEL
LIN {X 0,Y 580.214,Z 533.734,A -85,B 0,C 180,E1 -1881.292,E2 -1881.292} C_VEL
LIN {X 0,Y 580.13,Z 541.09,A -85,B 0,C 180,E1 -1882.692,E2 -1882.692} C_VEL
LIN {X 0,Y 580.131,Z 546.925,A -85,B 0,C 180,E1 -1884.09,E2 -1884.09} C_VEL
LIN {X 0,Y 580.041,Z 550.385,A -85,B 0,C 180,E1 -1885.135,E2 -1885.135} C_VEL
LIN {X 0,Y 580.104,Z 553.889,A -85,B 0,C 180,E1 -1886.527,E2 -1886.527} C_VEL
LIN {X 0,Y 580.039,Z 556.193,A -85,B 0,C 180,E1 -1887.917,E2 -1887.917} C_VEL
LIN {X 0,Y 580.038,Z 557.35,A -85,B 0,C 180,E1 -1889.306,E2 -1889.306} C_VEL
LIN {X 0,Y 580.038,Z 557.349,A -85,B 0,C 180,E1 -1890.695,E2 -1890.695} C_VEL
LIN {X 0,Y 580.039,Z 556.192,A -85,B 0,C 180,E1 -1892.083,E2 -1892.083} C_VEL
LIN {X 0,Y 580.104,Z 553.886,A -85,B 0,C 180,E1 -1893.473,E2 -1893.473} C_VEL
LIN {X 0,Y 580.041,Z 550.383,A -85,B 0,C 180,E1 -1894.866,E2 -1894.866} C_VEL
LIN {X 0,Y 580.093,Z 545.607,A -85,B 0,C 180,E1 -1896.26,E2 -1896.26} C_VEL
LIN {X 0,Y 580.165,Z 539.422,A -85,B 0,C 180,E1 -1897.658,E2 -1897.658} C_VEL
LIN {X 0,Y 580.207,Z 531.648,A -85,B 0,C 180,E1 -1899.06,E2 -1899.06} C_VEL
LIN {X 0,Y 580.309,Z 523.367,A -85,B 0,C 180,E1 -1900.29,E2 -1900.29} C_VEL
LIN {X 0,Y 580.383,Z 513.392,A -85,B 0,C 180,E1 -1901.525,E2 -1901.525} C_VEL
LIN {X 0,Y 580.541,Z 503.187,A -85,B 0,C 180,E1 -1902.586,E2 -1902.586} C_VEL
LIN {X 0,Y 580.674,Z 491.014,A -85,B 0,C 180,E1 -1903.652,E2 -1903.652} C_VEL
LIN {X 0,Y 580.847,Z 478.802,A -85,B 0,C 180,E1 -1904.542,E2 -1904.542} C_VEL
LIN {X 0,Y 580.996,Z 465.515,A -85,B 0,C 180,E1 -1905.344,E2 -1905.344} C_VEL
LIN {X 0,Y 581.153,Z 450.83,A -85,B 0,C 180,E1 -1906.06,E2 -1906.06} C_VEL
LIN {X 0,Y 581.347,Z 436.608,A -85,B 0,C 180,E1 -1906.595,E2 -1906.595} C_VEL
LIN {X 0,Y 581.45,Z 421.487,A -85,B 0,C 180,E1 -1907.018,E2 -1907.018} C_VEL
LIN {X 0,Y 581.363,Z 406.977,A -85,B 0,C 180,E1 -1907.293,E2 -1907.293} C_VEL
LIN {X 0,Y 580.192,Z 401.695,A -85,B 0,C 180,E1 -1907.415,E2 -1907.415} C_VEL
LIN {X 0,Y 580.266,Z 392.838,A -85,B 0,C 180,E1 -1910.193,E2 -1910.193} C_VEL
LIN {X 0,Y 580.297,Z 384.023,A -85,B 0,C 180,E1 -1913.01,E2 -1913.01} C_VEL
LIN {X 0,Y 580.361,Z 375.325,A -85,B 0,C 180,E1 -1915.846,E2 -1915.846} C_VEL
LIN {X 0,Y 580.45,Z 367.153,A -85,B 0,C 180,E1 -1918.572,E2 -1918.572} C_VEL
LIN {X 0,Y 580.461,Z 358.74,A -85,B 0,C 180,E1 -1921.375,E2 -1921.375} C_VEL
LIN {X 0,Y 580.521,Z 351.558,A -85,B 0,C 180,E1 -1923.841,E2 -1923.841} C_VEL
LIN {X 0,Y 580.586,Z 344.376,A -85,B 0,C 180,E1 -1926.381,E2 -1926.381} C_VEL
LIN {X 0,Y 580.618,Z 336.75,A -85,B 0,C 180,E1 -1929.224,E2 -1929.224} C_VEL
LIN {X 0,Y 580.632,Z 331.384,A -85,B 0,C 180,E1 -1931.371,E2 -1931.371} C_VEL
LIN {X 0,Y 580.323,Z 328.827,A -85,B 0,C 180,E1 -1932.556,E2 -1932.556} C_VEL
LIN {X 0,Y 580.272,Z 328.831,A -85,B 0,C 180,E1 -1935.609,E2 -1935.609} C_VEL
LIN {X 0,Y 580.283,Z 328.828,A -85,B 0,C 180,E1 -1938.232,E2 -1938.232} C_VEL
LIN {X 0,Y 580.288,Z 328.826,A -85,B 0,C 180,E1 -1940.966,E2 -1940.966} C_VEL
LIN {X 0,Y 580.299,Z 328.827,A -85,B 0,C 180,E1 -1943.599,E2 -1943.599} C_VEL
LIN {X 0,Y 580.32,Z 328.826,A -85,B 0,C 180,E1 -1946.146,E2 -1946.146} C_VEL
LIN {X 0,Y 580.278,Z 328.827,A -85,B 0,C 180,E1 -1948.615,E2 -1948.615} C_VEL
LIN {X 0,Y 580.295,Z 328.829,A -85,B 0,C 180,E1 -1951.024,E2 -1951.024} C_VEL
LIN {X 0,Y 580.292,Z 328.828,A -85,B 0,C 180,E1 -1953.667,E2 -1953.667} C_VEL
LIN {X 0,Y 580.301,Z 328.827,A -85,B 0,C 180,E1 -1955.684,E2 -1955.684} C_VEL
LIN {X 0,Y 580.288,Z 328.829,A -85,B 0,C 180,E1 -1958.695,E2 -1958.695} C_VEL
LIN {X 0,Y 580.304,Z 328.823,A -85,B 0,C 180,E1 -1960.914,E2 -1960.914} C_VEL
LIN {X 0,Y 580.283,Z 328.826,A -85,B 0,C 180,E1 -1963.826,E2 -1963.826} C_VEL
LIN {X 0,Y 580.331,Z 328.825,A -85,B 0,C 180,E1 -1965.983,E2 -1965.983} C_VEL
LIN {X 0,Y 580.309,Z 328.825,A -85,B 0,C 180,E1 -1968.827,E2 -1968.827} C_VEL
LIN {X 0,Y 580.331,Z 328.821,A -85,B 0,C 180,E1 -1971.644,E2 -1971.644} C_VEL
LIN {X 0,Y 580.324,Z 328.821,A -85,B 0,C 180,E1 -1974.44,E2 -1974.44} C_VEL
LIN {X 0,Y 580.346,Z 328.819,A -85,B 0,C 180,E1 -1977.224,E2 -1977.224} C_VEL
LIN {X 0,Y 580.354,Z 328.821,A -85,B 0,C 180,E1 -1980,E2 -1980} C_VEL
LIN {X 0,Y 580.348,Z 328.823,A -85,B 0,C 180,E1 -1982.777,E2 -1982.777} C_VEL
LIN {X 0,Y 580.329,Z 328.822,A -85,B 0,C 180,E1 -1985.56,E2 -1985.56} C_VEL
LIN {X 0,Y 580.336,Z 328.82,A -85,B 0,C 180,E1 -1988.356,E2 -1988.356} C_VEL
LIN {X 0,Y 580.304,Z 328.822,A -85,B 0,C 180,E1 -1991.191,E2 -1991.191} C_VEL
LIN {X 0,Y 580.329,Z 328.82,A -85,B 0,C 180,E1 -1994.017,E2 -1994.017} C_VEL
LIN {X 0,Y 580.316,Z 328.823,A -85,B 0,C 180,E1 -1996.914,E2 -1996.914} C_VEL
LIN {X 0,Y 580.308,Z 328.823,A -85,B 0,C 180,E1 -1999.822,E2 -1999.822} C_VEL
LIN {X 0,Y 580.287,Z 328.828,A -85,B 0,C 180,E1 -2001.328,E2 -2001.328} C_VEL
LIN {X 0,Y 579.588,Z 328.912,A -85,B 0,C 180,E1 -2001.907,E2 -2001.907} C_VEL
LIN {X 0,Y 576.71,Z 329.275,A -85,B 0,C 180,E1 -2002.847,E2 -2002.847} C_VEL
LIN {X 0,Y 574.315,Z 329.571,A -85,B 0,C 180,E1 -2003.603,E2 -2003.603} C_VEL
LIN {X 0,Y 573.318,Z 329.699,A -85,B 0,C 180,E1 -2004.187,E2 -2004.187} C_VEL
LIN {X 0,Y 573.252,Z 329.701,A -85,B 0,C 180,E1 -2004.385,E2 -2004.385} C_VEL
LIN {X 0,Y 573.255,Z 329.702,A -85,B 0,C 180,E1 -2006.976,E2 -2006.976} C_VEL
LIN {X 0,Y 573.251,Z 329.702,A -85,B 0,C 180,E1 -2009.488,E2 -2009.488} C_VEL
LIN {X 0,Y 573.257,Z 329.7,A -85,B 0,C 180,E1 -2012.645,E2 -2012.645} C_VEL
LIN {X 0,Y 573.258,Z 329.703,A -85,B 0,C 180,E1 -2015.184,E2 -2015.184} C_VEL
LIN {X 0,Y 573.24,Z 329.708,A -85,B 0,C 180,E1 -2017.807,E2 -2017.807} C_VEL
LIN {X 0,Y 573.273,Z 329.701,A -85,B 0,C 180,E1 -2020.528,E2 -2020.528} C_VEL
LIN {X 0,Y 573.248,Z 329.705,A -85,B 0,C 180,E1 -2023.669,E2 -2023.669} C_VEL
LIN {X 0,Y 573.244,Z 329.705,A -85,B 0,C 180,E1 -2026.641,E2 -2026.641} C_VEL
LIN {X 0,Y 573.205,Z 329.714,A -85,B 0,C 180,E1 -2028.54,E2 -2028.54} C_VEL
LIN {X 0,Y 573.152,Z 329.968,A -85,B 0,C 180,E1 -2029.486,E2 -2029.486} C_VEL
LIN {X 0,Y 573.151,Z 332.708,A -85,B 0,C 180,E1 -2032.186,E2 -2032.186} C_VEL
LIN {X 0,Y 573.102,Z 335.727,A -85,B 0,C 180,E1 -2035.248,E2 -2035.248} C_VEL
LIN {X 0,Y 573.074,Z 338.305,A -85,B 0,C 180,E1 -2037.8,E2 -2037.8} C_VEL
LIN {X 0,Y 573.062,Z 341.144,A -85,B 0,C 180,E1 -2040.545,E2 -2040.545} C_VEL
LIN {X 0,Y 573.011,Z 343.735,A -85,B 0,C 180,E1 -2043.012,E2 -2043.012} C_VEL
LIN {X 0,Y 573.004,Z 347.411,A -85,B 0,C 180,E1 -2046.124,E2 -2046.124} C_VEL
LIN {X 0,Y 572.983,Z 351.127,A -85,B 0,C 180,E1 -2049.163,E2 -2049.163} C_VEL
LIN {X 0,Y 572.967,Z 353.915,A -85,B 0,C 180,E1 -2051.402,E2 -2051.402} C_VEL
LIN {X 0,Y 572.962,Z 355.24,A -85,B 0,C 180,E1 -2052.456,E2 -2052.456} C_VEL
LIN {X 0,Y 574.757,Z 363.12,A -85,B 0,C 180,E1 -2052.646,E2 -2052.646} C_VEL
LIN {X 0,Y 574.609,Z 378.048,A -85,B 0,C 180,E1 -2052.984,E2 -2052.984} C_VEL
LIN {X 0,Y 574.43,Z 393.238,A -85,B 0,C 180,E1 -2053.48,E2 -2053.48} C_VEL
LIN {X 0,Y 574.235,Z 407.721,A -85,B 0,C 180,E1 -2054.107,E2 -2054.107} C_VEL
LIN {X 0,Y 574.026,Z 421.026,A -85,B 0,C 180,E1 -2054.829,E2 -2054.829} C_VEL
LIN {X 0,Y 573.86,Z 434.549,A -85,B 0,C 180,E1 -2055.728,E2 -2055.728} C_VEL
LIN {X 0,Y 573.63,Z 446.877,A -85,B 0,C 180,E1 -2056.719,E2 -2056.719} C_VEL
LIN {X 0,Y 573.459,Z 458.076,A -85,B 0,C 180,E1 -2057.795,E2 -2057.795} C_VEL
LIN {X 0,Y 573.295,Z 467.581,A -85,B 0,C 180,E1 -2058.877,E2 -2058.877} C_VEL
LIN {X 0,Y 573.203,Z 476.775,A -85,B 0,C 180,E1 -2060.116,E2 -2060.116} C_VEL
LIN {X 0,Y 573.134,Z 484.484,A -85,B 0,C 180,E1 -2061.36,E2 -2061.36} C_VEL
LIN {X 0,Y 573.076,Z 490.881,A -85,B 0,C 180,E1 -2062.601,E2 -2062.601} C_VEL
LIN {X 0,Y 573.042,Z 496.766,A -85,B 0,C 180,E1 -2064.016,E2 -2064.016} C_VEL
LIN {X 0,Y 572.949,Z 500.249,A -85,B 0,C 180,E1 -2065.074,E2 -2065.074} C_VEL
LIN {X 0,Y 573.004,Z 503.794,A -85,B 0,C 180,E1 -2066.484,E2 -2066.484} C_VEL
LIN {X 0,Y 572.938,Z 506.14,A -85,B 0,C 180,E1 -2067.891,E2 -2067.891} C_VEL
LIN {X 0,Y 572.936,Z 507.337,A -85,B 0,C 180,E1 -2069.297,E2 -2069.297} C_VEL
LIN {X 0,Y 572.937,Z 507.36,A -85,B 0,C 180,E1 -2070.703,E2 -2070.703} C_VEL
LIN {X 0,Y 572.939,Z 506.244,A -85,B 0,C 180,E1 -2072.109,E2 -2072.109} C_VEL
LIN {X 0,Y 573.006,Z 503.981,A -85,B 0,C 180,E1 -2073.516,E2 -2073.516} C_VEL
LIN {X 0,Y 572.949,Z 500.521,A -85,B 0,C 180,E1 -2074.925,E2 -2074.925} C_VEL
LIN {X 0,Y 573.007,Z 495.789,A -85,B 0,C 180,E1 -2076.337,E2 -2076.337} C_VEL
LIN {X 0,Y 573.094,Z 489.656,A -85,B 0,C 180,E1 -2077.752,E2 -2077.752} C_VEL
LIN {X 0,Y 573.134,Z 481.936,A -85,B 0,C 180,E1 -2079.172,E2 -2079.172} C_VEL
LIN {X 0,Y 573.265,Z 473.695,A -85,B 0,C 180,E1 -2080.418,E2 -2080.418} C_VEL
LIN {X 0,Y 573.354,Z 463.787,A -85,B 0,C 180,E1 -2081.668,E2 -2081.668} C_VEL
LIN {X 0,Y 573.534,Z 453.638,A -85,B 0,C 180,E1 -2082.742,E2 -2082.742} C_VEL
LIN {X 0,Y 573.721,Z 441.56,A -85,B 0,C 180,E1 -2083.82,E2 -2083.82} C_VEL
LIN {X 0,Y 573.94,Z 428.693,A -85,B 0,C 180,E1 -2084.773,E2 -2084.773} C_VEL
LIN {X 0,Y 574.149,Z 414.722,A -85,B 0,C 180,E1 -2085.622,E2 -2085.622} C_VEL
LIN {X 0,Y 574.339,Z 399.789,A -85,B 0,C 180,E1 -2086.346,E2 -2086.346} C_VEL
LIN {X 0,Y 574.541,Z 385.281,A -85,B 0,C 180,E1 -2086.889,E2 -2086.889} C_VEL
LIN {X 0,Y 574.704,Z 369.398,A -85,B 0,C 180,E1 -2087.319,E2 -2087.319} C_VEL
LIN {X 0,Y 574.499,Z 361.858,A -85,B 0,C 180,E1 -2087.476,E2 -2087.476} C_VEL
LIN {X 0,Y 572.971,Z 355.245,A -85,B 0,C 180,E1 -2087.629,E2 -2087.629} C_VEL
LIN {X 0,Y 572.983,Z 352.169,A -85,B 0,C 180,E1 -2090.086,E2 -2090.086} C_VEL
LIN {X 0,Y 572.987,Z 348.45,A -85,B 0,C 180,E1 -2093.11,E2 -2093.11} C_VEL
LIN {X 0,Y 573.002,Z 345.661,A -85,B 0,C 180,E1 -2095.422,E2 -2095.422} C_VEL
LIN {X 0,Y 573.036,Z 342.822,A -85,B 0,C 180,E1 -2097.988,E2 -2097.988} C_VEL
LIN {X 0,Y 573.08,Z 339.633,A -85,B 0,C 180,E1 -2101.002,E2 -2101.002} C_VEL
LIN {X 0,Y 573.121,Z 337.064,A -85,B 0,C 180,E1 -2103.502,E2 -2103.502} C_VEL
LIN {X 0,Y 573.115,Z 334.521,A -85,B 0,C 180,E1 -2106.058,E2 -2106.058} C_VEL
LIN {X 0,Y 573.154,Z 331.891,A -85,B 0,C 180,E1 -2108.708,E2 -2108.708} C_VEL
LIN {X 0,Y 573.149,Z 330.041,A -85,B 0,C 180,E1 -2110.533,E2 -2110.533} C_VEL
LIN {X 0,Y 573.242,Z 329.703,A -85,B 0,C 180,E1 -2112.4,E2 -2112.4} C_VEL
LIN {X 0,Y 573.227,Z 329.71,A -85,B 0,C 180,E1 -2114.675,E2 -2114.675} C_VEL
LIN {X 0,Y 573.239,Z 329.709,A -85,B 0,C 180,E1 -2117.599,E2 -2117.599} C_VEL
LIN {X 0,Y 573.248,Z 329.705,A -85,B 0,C 180,E1 -2120.393,E2 -2120.393} C_VEL
LIN {X 0,Y 573.256,Z 329.701,A -85,B 0,C 180,E1 -2123.078,E2 -2123.078} C_VEL
LIN {X 0,Y 573.273,Z 329.699,A -85,B 0,C 180,E1 -2125.672,E2 -2125.672} C_VEL
LIN {X 0,Y 573.248,Z 329.706,A -85,B 0,C 180,E1 -2128.185,E2 -2128.185} C_VEL
LIN {X 0,Y 573.267,Z 329.7,A -85,B 0,C 180,E1 -2130.634,E2 -2130.634} C_VEL
LIN {X 0,Y 573.269,Z 329.698,A -85,B 0,C 180,E1 -2133.5,E2 -2133.5} C_VEL
LIN {X 0,Y 573.233,Z 329.707,A -85,B 0,C 180,E1 -2136.134,E2 -2136.134} C_VEL
LIN {X 0,Y 573.25,Z 329.702,A -85,B 0,C 180,E1 -2139.173,E2 -2139.173} C_VEL
LIN {X 0,Y 573.236,Z 329.703,A -85,B 0,C 180,E1 -2141.412,E2 -2141.412} C_VEL
LIN {X 0,Y 573.258,Z 329.705,A -85,B 0,C 180,E1 -2143.622,E2 -2143.622} C_VEL
LIN {X 0,Y 573.272,Z 329.697,A -85,B 0,C 180,E1 -2145.807,E2 -2145.807} C_VEL
LIN {X 0,Y 573.261,Z 329.7,A -85,B 0,C 180,E1 -2148.745,E2 -2148.745} C_VEL
LIN {X 0,Y 573.289,Z 329.698,A -85,B 0,C 180,E1 -2151.54,E2 -2151.54} C_VEL
LIN {X 0,Y 573.295,Z 329.7,A -85,B 0,C 180,E1 -2154.372,E2 -2154.372} C_VEL
LIN {X 0,Y 573.305,Z 329.695,A -85,B 0,C 180,E1 -2157.892,E2 -2157.892} C_VEL
LIN {X 0,Y 573.332,Z 329.693,A -85,B 0,C 180,E1 -2160.702,E2 -2160.702} C_VEL
LIN {X 0,Y 573.239,Z 329.706,A -85,B 0,C 180,E1 -2163.514,E2 -2163.514} C_VEL
LIN {X 0,Y 573.291,Z 329.697,A -85,B 0,C 180,E1 -2165.628,E2 -2165.628} C_VEL
LIN {X 0,Y 573.284,Z 329.698,A -85,B 0,C 180,E1 -2168.459,E2 -2168.459} C_VEL
LIN {X 0,Y 573.298,Z 329.697,A -85,B 0,C 180,E1 -2171.311,E2 -2171.311} C_VEL
LIN {X 0,Y 573.281,Z 329.699,A -85,B 0,C 180,E1 -2174.425,E2 -2174.425} C_VEL
LIN {X 0,Y 573.257,Z 329.705,A -85,B 0,C 180,E1 -2177.112,E2 -2177.112} C_VEL
LIN {X 0,Y 573.251,Z 329.707,A -85,B 0,C 180,E1 -2180.077,E2 -2180.077} C_VEL
LIN {X 0,Y 573.232,Z 329.71,A -85,B 0,C 180,E1 -2183.099,E2 -2183.099} C_VEL
LIN {X 0,Y 573.252,Z 329.702,A -85,B 0,C 180,E1 -2185.41,E2 -2185.41} C_VEL
LIN {X 0,Y 573.251,Z 329.704,A -85,B 0,C 180,E1 -2188.03,E2 -2188.03} C_VEL
LIN {X 0,Y 573.243,Z 329.706,A -85,B 0,C 180,E1 -2190.885,E2 -2190.885} C_VEL
LIN {X 0,Y 573.26,Z 329.705,A -85,B 0,C 180,E1 -2193.524,E2 -2193.524} C_VEL
LIN {X 0,Y 573.26,Z 329.701,A -85,B 0,C 180,E1 -2196.048,E2 -2196.048} C_VEL
LIN {X 0,Y 573.249,Z 329.704,A -85,B 0,C 180,E1 -2198.701,E2 -2198.701} C_VEL
LIN {X 0,Y 573.253,Z 329.705,A -85,B 0,C 180,E1 -2201.596,E2 -2201.596} C_VEL
LIN {X 0,Y 573.234,Z 329.708,A -85,B 0,C 180,E1 -2204.334,E2 -2204.334} C_VEL
LIN {X 0,Y 573.301,Z 329.894,A -85,B 0,C 180,E1 -2207.352,E2 -2207.352} C_VEL
LIN {X 0,Y 573.758,Z 333.779,A -85,B 0,C 180,E1 -2209.042,E2 -2209.042} C_VEL
LIN {X 0,Y 573.633,Z 340.328,A -85,B 0,C 180,E1 -2211.638,E2 -2211.638} C_VEL
LIN {X 0,Y 573.543,Z 347.81,A -85,B 0,C 180,E1 -2214.406,E2 -2214.406} C_VEL
LIN {X 0,Y 573.485,Z 354.997,A -85,B 0,C 180,E1 -2216.952,E2 -2216.952} C_VEL
LIN {X 0,Y 573.454,Z 362.269,A -85,B 0,C 180,E1 -2219.458,E2 -2219.458} C_VEL
LIN {X 0,Y 573.397,Z 369.743,A -85,B 0,C 180,E1 -2221.944,E2 -2221.944} C_VEL
LIN {X 0,Y 573.361,Z 377.662,A -85,B 0,C 180,E1 -2224.595,E2 -2224.595} C_VEL
LIN {X 0,Y 573.259,Z 385.835,A -85,B 0,C 180,E1 -2227.283,E2 -2227.283} C_VEL
LIN {X 0,Y 573.214,Z 394.008,A -85,B 0,C 180,E1 -2229.922,E2 -2229.922} C_VEL
LIN {X 0,Y 573.149,Z 401.731,A -85,B 0,C 180,E1 -2232.376,E2 -2232.376} C_VEL
LIN {X 0,Y 574.708,Z 408.536,A -85,B 0,C 180,E1 -2232.525,E2 -2232.525} C_VEL
LIN {X 0,Y 574.604,Z 424.086,A -85,B 0,C 180,E1 -2232.838,E2 -2232.838} C_VEL
LIN {X 0,Y 574.506,Z 439.217,A -85,B 0,C 180,E1 -2233.293,E2 -2233.293} C_VEL
LIN {X 0,Y 574.278,Z 452.829,A -85,B 0,C 180,E1 -2233.835,E2 -2233.835} C_VEL
LIN {X 0,Y 574.088,Z 467.108,A -85,B 0,C 180,E1 -2234.558,E2 -2234.558} C_VEL
LIN {X 0,Y 573.884,Z 480.418,A -85,B 0,C 180,E1 -2235.392,E2 -2235.392} C_VEL
LIN {X 0,Y 573.689,Z 493.167,A -85,B 0,C 180,E1 -2236.36,E2 -2236.36} C_VEL
LIN {X 0,Y 573.511,Z 504.974,A -85,B 0,C 180,E1 -2237.437,E2 -2237.437} C_VEL
LIN {X 0,Y 573.348,Z 514.904,A -85,B 0,C 180,E1 -2238.511,E2 -2238.511} C_VEL
LIN {X 0,Y 573.256,Z 524.622,A -85,B 0,C 180,E1 -2239.761,E2 -2239.761} C_VEL
LIN {X 0,Y 573.135,Z 532.723,A -85,B 0,C 180,E1 -2241.005,E2 -2241.005} C_VEL
LIN {X 0,Y 573.093,Z 539.426,A -85,B 0,C 180,E1 -2242.248,E2 -2242.248} C_VEL
LIN {X 0,Y 573.015,Z 545.608,A -85,B 0,C 180,E1 -2243.663,E2 -2243.663} C_VEL
LIN {X 0,Y 572.951,Z 550.386,A -85,B 0,C 180,E1 -2245.075,E2 -2245.075} C_VEL
LIN {X 0,Y 573.004,Z 553.889,A -85,B 0,C 180,E1 -2246.484,E2 -2246.484} C_VEL
LIN {X 0,Y 572.938,Z 556.193,A -85,B 0,C 180,E1 -2247.891,E2 -2247.891} C_VEL
LIN {X 0,Y 572.938,Z 557.349,A -85,B 0,C 180,E1 -2249.297,E2 -2249.297} C_VEL
LIN {X 0,Y 572.938,Z 557.349,A -85,B 0,C 180,E1 -2250.703,E2 -2250.703} C_VEL
LIN {X 0,Y 572.938,Z 556.191,A -85,B 0,C 180,E1 -2252.109,E2 -2252.109} C_VEL
LIN {X 0,Y 573.004,Z 553.886,A -85,B 0,C 180,E1 -2253.516,E2 -2253.516} C_VEL
LIN {X 0,Y 572.951,Z 550.384,A -85,B 0,C 180,E1 -2254.926,E2 -2254.926} C_VEL
LIN {X 0,Y 573.014,Z 545.607,A -85,B 0,C 180,E1 -2256.338,E2 -2256.338} C_VEL
LIN {X 0,Y 573.093,Z 539.422,A -85,B 0,C 180,E1 -2257.753,E2 -2257.753} C_VEL
LIN {X 0,Y 573.136,Z 531.647,A -85,B 0,C 180,E1 -2259.173,E2 -2259.173} C_VEL
LIN {X 0,Y 573.27,Z 523.367,A -85,B 0,C 180,E1 -2260.418,E2 -2260.418} C_VEL
LIN {X 0,Y 573.386,Z 513.389,A -85,B 0,C 180,E1 -2261.668,E2 -2261.668} C_VEL
LIN {X 0,Y 573.568,Z 503.187,A -85,B 0,C 180,E1 -2262.742,E2 -2262.742} C_VEL
LIN {X 0,Y 573.703,Z 491.015,A -85,B 0,C 180,E1 -2263.821,E2 -2263.821} C_VEL
LIN {X 0,Y 573.963,Z 477.897,A -85,B 0,C 180,E1 -2264.781,E2 -2264.781} C_VEL
LIN {X 0,Y 574.136,Z 465.513,A -85,B 0,C 180,E1 -2265.532,E2 -2265.532} C_VEL
LIN {X 0,Y 574.326,Z 450.827,A -85,B 0,C 180,E1 -2266.256,E2 -2266.256} C_VEL
LIN {X 0,Y 574.547,Z 436.607,A -85,B 0,C 180,E1 -2266.798,E2 -2266.798} C_VEL
LIN {X 0,Y 574.666,Z 421.713,A -85,B 0,C 180,E1 -2267.22,E2 -2267.22} C_VEL
LIN {X 0,Y 574.589,Z 408.064,A -85,B 0,C 180,E1 -2267.486,E2 -2267.486} C_VEL
LIN {X 0,Y 573.157,Z 401.667,A -85,B 0,C 180,E1 -2267.644,E2 -2267.644} C_VEL
LIN {X 0,Y 573.22,Z 392.838,A -85,B 0,C 180,E1 -2270.452,E2 -2270.452} C_VEL
LIN {X 0,Y 573.282,Z 383.499,A -85,B 0,C 180,E1 -2273.48,E2 -2273.48} C_VEL
LIN {X 0,Y 573.355,Z 375.325,A -85,B 0,C 180,E1 -2276.186,E2 -2276.186} C_VEL
LIN {X 0,Y 573.469,Z 365.819,A -85,B 0,C 180,E1 -2279.355,E2 -2279.355} C_VEL
LIN {X 0,Y 573.51,Z 357.214,A -85,B 0,C 180,E1 -2282.269,E2 -2282.269} C_VEL
LIN {X 0,Y 573.544,Z 348.99,A -85,B 0,C 180,E1 -2285.164,E2 -2285.164} C_VEL
LIN {X 0,Y 573.606,Z 341.848,A -85,B 0,C 180,E1 -2287.779,E2 -2287.779} C_VEL
LIN {X 0,Y 573.719,Z 334.706,A -85,B 0,C 180,E1 -2290.581,E2 -2290.581} C_VEL
LIN {X 0,Y 573.638,Z 332.168,A -85,B 0,C 180,E1 -2291.639,E2 -2291.639} C_VEL
LIN {X 0,Y 573.273,Z 329.704,A -85,B 0,C 180,E1 -2292.779,E2 -2292.779} C_VEL
LIN {X 0,Y 573.238,Z 329.707,A -85,B 0,C 180,E1 -2295.667,E2 -2295.667} C_VEL
LIN {X 0,Y 573.234,Z 329.709,A -85,B 0,C 180,E1 -2298.543,E2 -2298.543} C_VEL
LIN {X 0,Y 573.249,Z 329.704,A -85,B 0,C 180,E1 -2301.299,E2 -2301.299} C_VEL
LIN {X 0,Y 573.267,Z 329.701,A -85,B 0,C 180,E1 -2304.011,E2 -2304.011} C_VEL
LIN {X 0,Y 573.272,Z 329.703,A -85,B 0,C 180,E1 -2306.518,E2 -2306.518} C_VEL
LIN {X 0,Y 573.232,Z 329.708,A -85,B 0,C 180,E1 -2309.118,E2 -2309.118} C_VEL
LIN {X 0,Y 573.255,Z 329.703,A -85,B 0,C 180,E1 -2311.971,E2 -2311.971} C_VEL
LIN {X 0,Y 573.251,Z 329.702,A -85,B 0,C 180,E1 -2314.59,E2 -2314.59} C_VEL
